   1:  PR[91,2] = PR[90,2] + -6.880;
   1:L PR[91] R[100]mm/sec CNT100;
   1:  PR[91,1] = PR[90,1] + -40.976;
   1:  PR[91,2] = PR[90,2] + -9.031;
   1:L PR[91] R[100]mm/sec CNT100;
   1:  PR[91,1] = PR[90,1] + -40.215;
   1:  PR[91,2] = PR[90,2] + -10.350;
   1:L PR[91] R[100]mm/sec CNT100;
   1:  PR[91,1] = PR[90,1] + -38.856;
   1:  PR[91,2] = PR[90,2] + -12.292;
   1:L PR[91] R[100]mm/sec CNT100;
   1:  PR[91,1] = PR[90,1] + -37.178;
   1:  PR[91,2] = PR[90,2] + -13.971;
   1:L PR[91] R[100]mm/sec CNT100;
   1:  PR[91,1] = PR[90,1] + -36.012;
   1:  PR[91,2] = PR[90,2] + -14.949;
   1:L PR[91] R[100]mm/sec CNT100;
   1:  PR[91,1] = PR[90,1] + -34.070;
   1:  PR[91,2] = PR[90,2] + -16.309;
   1:L PR[91] R[100]mm/sec CNT100;
   1:  PR[91,1] = PR[90,1] + -31.919;
   1:  PR[91,2] = PR[90,2] + -17.313;
   1:L PR[91] R[100]mm/sec CNT100;
   1:  PR[91,1] = PR[90,1] + -30.489;
   1:  PR[91,2] = PR[90,2] + -17.834;
   1:L PR[91] R[100]mm/sec CNT100;
   1:  PR[91,1] = PR[90,1] + -28.198;
   1:  PR[91,2] = PR[90,2] + -18.448;
   1:L PR[91] R[100]mm/sec CNT100;
   1:  PR[91,1] = PR[90,1] + -25.833;
   1:  PR[91,2] = PR[90,2] + -18.655;
   1:L PR[91] R[100]mm/sec CNT100;
   1:  PR[91,1] = PR[90,1] + -24.309;
   1:L PR[91] R[100]mm/sec CNT100;
   1:  PR[91,1] = PR[90,1] + -22.033;
   1:  PR[91,2] = PR[90,2] + -18.456;
   1:L PR[91] R[100]mm/sec CNT100;
   1:  PR[91,1] = PR[90,1] + -20.603;
   1:  PR[91,2] = PR[90,2] + -17.935;
   1:L PR[91] R[100]mm/sec CNT100;
   1:  PR[91,1] = PR[90,1] + -18.143;
   1:  PR[91,2] = PR[90,2] + -17.276;
   1:L PR[91] R[100]mm/sec CNT100;
   1:  PR[91,1] = PR[90,1] + -16.152;
   1:  PR[91,2] = PR[90,2] + -16.347;
   1:L PR[91] R[100]mm/sec CNT100;
   1:  PR[91,1] = PR[90,1] + -14.987;
   1:  PR[91,2] = PR[90,2] + -15.369;
   1:L PR[91] R[100]mm/sec CNT100;
   1:  PR[91,1] = PR[90,1] + -12.902;
   1:  PR[91,2] = PR[90,2] + -13.909;
   1:L PR[91] R[100]mm/sec CNT100;
   1:  PR[91,1] = PR[90,1] + -11.349;
   1:  PR[91,2] = PR[90,2] + -12.355;
   1:L PR[91] R[100]mm/sec CNT100;
   1:  PR[91,1] = PR[90,1] + -10.588;
   1:  PR[91,2] = PR[90,2] + -11.038;
   1:L PR[91] R[100]mm/sec CNT100;
   1:  PR[91,1] = PR[90,1] + -9.128;
   1:  PR[91,2] = PR[90,2] + -8.953;
   1:L PR[91] R[100]mm/sec CNT100;
   1:  PR[91,1] = PR[90,1] + -8.200;
   1:  PR[91,2] = PR[90,2] + -6.961;
   1:L PR[91] R[100]mm/sec CNT100;
   1:  PR[91,1] = PR[90,1] + -7.935;
   1:  PR[91,2] = PR[90,2] + -5.462;
   1:L PR[91] R[100]mm/sec CNT100;
   1:  PR[91,1] = PR[90,1] + -7.277;
   1:  PR[91,2] = PR[90,2] + -3.003;
   1:L PR[91] R[100]mm/sec CNT100;
   1:  PR[91,1] = PR[90,1] + -7.086;
   1:  PR[91,2] = PR[90,2] + -0.818;
   1:L PR[91] R[100]mm/sec CNT100;
   1:  PR[91,1] = PR[90,1] + -7.350;
   1:  PR[91,2] = PR[90,2] + 0.681;
   1:L PR[91] R[100]mm/sec CNT100;
   1:  PR[91,1] = PR[90,1] + -7.572;
   1:  PR[91,2] = PR[90,2] + 3.215;
   1:L PR[91] R[100]mm/sec CNT100;
   1:  PR[91,1] = PR[90,1] + -8.162;
   1:  PR[91,2] = PR[90,2] + 5.422;
   1:L PR[91] R[100]mm/sec CNT100;
   1:  PR[91,1] = PR[90,1] + -9.165;
   1:  PR[91,2] = PR[90,2] + 7.572;
   1:L PR[91] R[100]mm/sec CNT100;
   1:  PR[91,1] = PR[90,1] + -9.926;
   1:  PR[91,2] = PR[90,2] + 8.891;
   1:L PR[91] R[100]mm/sec CNT100;
   1:  PR[91,1] = PR[90,1] + -11.286;
   1:  PR[91,2] = PR[90,2] + 10.833;
   1:L PR[91] R[100]mm/sec CNT100;
   1:  PR[91,1] = PR[90,1] + -12.964;
   1:  PR[91,2] = PR[90,2] + 12.512;
   1:L PR[91] R[100]mm/sec CNT100;
   1:  PR[91,1] = PR[90,1] + -14.129;
   1:  PR[91,2] = PR[90,2] + 13.490;
   1:L PR[91] R[100]mm/sec CNT100;
   1:  PR[91,1] = PR[90,1] + -16.071;
   1:  PR[91,2] = PR[90,2] + 14.850;
   1:L PR[91] R[100]mm/sec CNT100;
   1:  PR[91,1] = PR[90,1] + -18.222;
   1:  PR[91,2] = PR[90,2] + 15.854;
   1:L PR[91] R[100]mm/sec CNT100;
   1:  PR[91,1] = PR[90,1] + -19.653;
   1:  PR[91,2] = PR[90,2] + 16.375;
   1:L PR[91] R[100]mm/sec CNT100;
   1:  PR[91,1] = PR[90,1] + -21.944;
   1:  PR[91,2] = PR[90,2] + 16.989;
   1:L PR[91] R[100]mm/sec CNT100;
   1:  PR[91,1] = PR[90,1] + -24.308;
   1:  PR[91,2] = PR[90,2] + 17.196;
   1:L PR[91] R[100]mm/sec CNT100;
   1:  PR[91,1] = PR[90,1] + -25.832;
   1:L PR[91] R[100]mm/sec CNT100;
   1:  PR[91,1] = PR[90,1] + -28.109;
   1:  PR[91,2] = PR[90,2] + 16.997;
   1:L PR[91] R[100]mm/sec CNT100;
   1:  PR[91,1] = PR[90,1] + -29.538;
   1:  PR[91,2] = PR[90,2] + 16.476;
   1:L PR[91] R[100]mm/sec CNT100;
   1:  PR[91,1] = PR[90,1] + -31.998;
   1:  PR[91,2] = PR[90,2] + 15.817;
   1:L PR[91] R[100]mm/sec CNT100;
   1:  PR[91,1] = PR[90,1] + -33.989;
   1:  PR[91,2] = PR[90,2] + 14.888;
   1:L PR[91] R[100]mm/sec CNT100;
   1:  PR[91,1] = PR[90,1] + -35.154;
   1:  PR[91,2] = PR[90,2] + 13.911;
   1:L PR[91] R[100]mm/sec CNT100;
   1:  PR[91,1] = PR[90,1] + -37.239;
   1:  PR[91,2] = PR[90,2] + 12.451;
   1:L PR[91] R[100]mm/sec CNT100;
   1:  PR[91,1] = PR[90,1] + -38.793;
   1:  PR[91,2] = PR[90,2] + 10.896;
   1:L PR[91] R[100]mm/sec CNT100;
   1:  PR[91,1] = PR[90,1] + -39.553;
   1:  PR[91,2] = PR[90,2] + 9.579;
   1:L PR[91] R[100]mm/sec CNT100;
   1:  PR[91,1] = PR[90,1] + -41.013;
   1:  PR[91,2] = PR[90,2] + 7.494;
   1:L PR[91] R[100]mm/sec CNT100;
   1:  PR[91,1] = PR[90,1] + -41.941;
   1:  PR[91,2] = PR[90,2] + 5.502;
   1:L PR[91] R[100]mm/sec CNT100;
   1:  PR[91,1] = PR[90,1] + -42.206;
   1:  PR[91,2] = PR[90,2] + 4.003;
   1:L PR[91] R[100]mm/sec CNT100;
   1:  PR[91,1] = PR[90,1] + -42.864;
   1:  PR[91,2] = PR[90,2] + 1.544;
   1:L PR[91] R[100]mm/sec CNT100;
   1:  PR[91,1] = PR[90,1] + -43.055;
   1:  PR[91,2] = PR[90,2] + -0.641;
   1:L PR[91] R[100]mm/sec CNT100;
   1:  PR[91,1] = PR[90,1] + -42.791;
   1:  PR[91,2] = PR[90,2] + -2.140;
   1:L PR[91] R[100]mm/sec CNT100TB   .50sec,CALL END_PUD;
   1:  PR[92] = PR[91];
   1:  PR[92,3] = PR[92,3] + 20;
   1:J PR[92] 10% FINE;
   1:  PR[91,1] = PR[90,1] + 29.399;
   1:  PR[91,2] = PR[90,2] + -17.935;
   1:  PR[92] = PR[91];
   1:  PR[92,3] = PR[92,3] + 20;
   1:J PR[92] 10% FINE;
   1:L PR[91] R[100]mm/sec CNT100;
   1:  CALL LASER_DRAHT_START;
   1:  PR[91,1] = PR[90,1] + 31.859;
   1:  PR[91,2] = PR[90,2] + -17.275;
   1:L PR[91] R[100]mm/sec CNT100;
   1:  PR[91,1] = PR[90,1] + 33.925;
   1:  PR[91,2] = PR[90,2] + -16.311;
   1:L PR[91] R[100]mm/sec CNT100;
   1:  PR[91,1] = PR[90,1] + 35.871;
   1:  PR[91,2] = PR[90,2] + -14.949;
   1:L PR[91] R[100]mm/sec CNT100;
   1:  PR[91,1] = PR[90,1] + 37.037;
   1:  PR[91,2] = PR[90,2] + -13.970;
   1:L PR[91] R[100]mm/sec CNT100;
   1:  PR[91,1] = PR[90,1] + 38.711;
   1:  PR[91,2] = PR[90,2] + -12.296;
   1:L PR[91] R[100]mm/sec CNT100;
   1:  PR[91,1] = PR[90,1] + 40.074;
   1:  PR[91,2] = PR[90,2] + -10.349;
   1:L PR[91] R[100]mm/sec CNT100;
   1:  PR[91,1] = PR[90,1] + 40.835;
   1:  PR[91,2] = PR[90,2] + -9.031;
   1:L PR[91] R[100]mm/sec CNT100;
   1:  PR[91,1] = PR[90,1] + 41.799;
   1:  PR[91,2] = PR[90,2] + -6.963;
   1:L PR[91] R[100]mm/sec CNT100;
   1:  PR[91,1] = PR[90,1] + 42.064;
   1:  PR[91,2] = PR[90,2] + -5.465;
   1:L PR[91] R[100]mm/sec CNT100;
   1:  PR[91,1] = PR[90,1] + 42.723;
   1:  PR[91,2] = PR[90,2] + -3.002;
   1:L PR[91] R[100]mm/sec CNT100;
   1:  PR[91,1] = PR[90,1] + 42.914;
   1:  PR[91,2] = PR[90,2] + -0.818;
   1:L PR[91] R[100]mm/sec CNT100;
   1:  PR[91,1] = PR[90,1] + 42.650;
   1:  PR[91,2] = PR[90,2] + 0.681;
   1:L PR[91] R[100]mm/sec CNT100;
   1:  PR[91,1] = PR[90,1] + 42.428;
   1:  PR[91,2] = PR[90,2] + 3.215;
   1:L PR[91] R[100]mm/sec CNT100;
   1:  PR[91,1] = PR[90,1] + 41.859;
   1:  PR[91,2] = PR[90,2] + 5.341;
   1:L PR[91] R[100]mm/sec CNT100;
   1:  PR[91,1] = PR[90,1] + 41.098;
   1:  PR[91,2] = PR[90,2] + 6.658;
   1:L PR[91] R[100]mm/sec CNT100;
   1:  PR[91,1] = PR[90,1] + 40.022;
   1:  PR[91,2] = PR[90,2] + 8.965;
   1:L PR[91] R[100]mm/sec CNT100;
   1:  PR[91,1] = PR[90,1] + 38.759;
   1:  PR[91,2] = PR[90,2] + 10.768;
   1:L PR[91] R[100]mm/sec CNT100;
   1:  PR[91,1] = PR[90,1] + 37.594;
   1:  PR[91,2] = PR[90,2] + 11.746;
   1:L PR[91] R[100]mm/sec CNT100;
   1:  PR[91,1] = PR[90,1] + 35.795;
   1:  PR[91,2] = PR[90,2] + 13.543;
   1:L PR[91] R[100]mm/sec CNT100;
   1:  PR[91,1] = PR[90,1] + 33.992;
   1:  PR[91,2] = PR[90,2] + 14.805;
   1:L PR[91] R[100]mm/sec CNT100;
   1:  PR[91,1] = PR[90,1] + 32.563;
   1:  PR[91,2] = PR[90,2] + 15.325;
   1:L PR[91] R[100]mm/sec CNT100;
   1:  PR[91,1] = PR[90,1] + 30.258;
   1:  PR[91,2] = PR[90,2] + 16.399;
   1:L PR[91] R[100]mm/sec CNT100;
   1:  PR[91,1] = PR[90,1] + 28.134;
   1:  PR[91,2] = PR[90,2] + 16.968;
   1:L PR[91] R[100]mm/sec CNT100;
   1:  PR[91,1] = PR[90,1] + 26.611;
   1:L PR[91] R[100]mm/sec CNT100;
   1:  PR[91,1] = PR[90,1] + 24.075;
   1:  PR[91,2] = PR[90,2] + 17.189;
   1:L PR[91] R[100]mm/sec CNT100;
   1:  PR[91,1] = PR[90,1] + 21.889;
   1:  PR[91,2] = PR[90,2] + 16.997;
   1:L PR[91] R[100]mm/sec CNT100;
   1:  PR[91,1] = PR[90,1] + 20.460;
   1:  PR[91,2] = PR[90,2] + 16.476;
   1:L PR[91] R[100]mm/sec CNT100;
   1:  PR[91,1] = PR[90,1] + 17.999;
   1:  PR[91,2] = PR[90,2] + 15.816;
   1:L PR[91] R[100]mm/sec CNT100;
   1:  PR[91,1] = PR[90,1] + 15.933;
   1:  PR[91,2] = PR[90,2] + 14.852;
   1:L PR[91] R[100]mm/sec CNT100;
   1:  PR[91,1] = PR[90,1] + 13.988;
   1:  PR[91,2] = PR[90,2] + 13.490;
   1:L PR[91] R[100]mm/sec CNT100;
   1:  PR[91,1] = PR[90,1] + 12.822;
   1:  PR[91,2] = PR[90,2] + 12.512;
   1:L PR[91] R[100]mm/sec CNT100;
   1:  PR[91,1] = PR[90,1] + 11.148;
   1:  PR[91,2] = PR[90,2] + 10.838;
   1:L PR[91] R[100]mm/sec CNT100;
   1:  PR[91,1] = PR[90,1] + 9.785;
   1:  PR[91,2] = PR[90,2] + 8.891;
   1:L PR[91] R[100]mm/sec CNT100;
   1:  PR[91,1] = PR[90,1] + 9.024;
   1:  PR[91,2] = PR[90,2] + 7.572;
   1:L PR[91] R[100]mm/sec CNT100;
   1:  PR[91,1] = PR[90,1] + 8.060;
   1:  PR[91,2] = PR[90,2] + 5.505;
   1:L PR[91] R[100]mm/sec CNT100;
   1:  PR[91,1] = PR[90,1] + 7.795;
   1:  PR[91,2] = PR[90,2] + 4.006;
   1:L PR[91] R[100]mm/sec CNT100;
   1:  PR[91,1] = PR[90,1] + 7.136;
   1:  PR[91,2] = PR[90,2] + 1.543;
   1:L PR[91] R[100]mm/sec CNT100;
   1:  PR[91,1] = PR[90,1] + 6.945;
   1:  PR[91,2] = PR[90,2] + -0.641;
   1:L PR[91] R[100]mm/sec CNT100;
   1:  PR[91,1] = PR[90,1] + 7.209;
   1:  PR[91,2] = PR[90,2] + -2.140;
   1:L PR[91] R[100]mm/sec CNT100;
   1:  PR[91,1] = PR[90,1] + 7.431;
   1:  PR[91,2] = PR[90,2] + -4.674;
   1:L PR[91] R[100]mm/sec CNT100;
   1:  PR[91,1] = PR[90,1] + 8.000;
   1:  PR[91,2] = PR[90,2] + -6.799;
   1:L PR[91] R[100]mm/sec CNT100;
   1:  PR[91,1] = PR[90,1] + 8.761;
   1:  PR[91,2] = PR[90,2] + -8.116;
   1:L PR[91] R[100]mm/sec CNT100;
   1:  PR[91,1] = PR[90,1] + 9.837;
   1:  PR[91,2] = PR[90,2] + -10.424;
   1:L PR[91] R[100]mm/sec CNT100;
   1:  PR[91,1] = PR[90,1] + 11.100;
   1:  PR[91,2] = PR[90,2] + -12.227;
   1:L PR[91] R[100]mm/sec CNT100;
   1:  PR[91,1] = PR[90,1] + 12.265;
   1:  PR[91,2] = PR[90,2] + -13.205;
   1:L PR[91] R[100]mm/sec CNT100;
   1:  PR[91,1] = PR[90,1] + 14.064;
   1:  PR[91,2] = PR[90,2] + -15.002;
   1:L PR[91] R[100]mm/sec CNT100;
   1:  PR[91,1] = PR[90,1] + 15.866;
   1:  PR[91,2] = PR[90,2] + -16.264;
   1:L PR[91] R[100]mm/sec CNT100;
   1:  PR[91,1] = PR[90,1] + 17.296;
   1:  PR[91,2] = PR[90,2] + -16.784;
   1:L PR[91] R[100]mm/sec CNT100;
   1:  PR[91,1] = PR[90,1] + 19.601;
   1:  PR[91,2] = PR[90,2] + -17.858;
   1:L PR[91] R[100]mm/sec CNT100;
   1:  PR[91,1] = PR[90,1] + 21.725;
   1:  PR[91,2] = PR[90,2] + -18.427;
   1:L PR[91] R[100]mm/sec CNT100;
   1:  PR[91,1] = PR[90,1] + 23.247;
   1:L PR[91] R[100]mm/sec CNT100;
   1:  PR[91,1] = PR[90,1] + 25.783;
   1:  PR[91,2] = PR[90,2] + -18.647;
   1:L PR[91] R[100]mm/sec CNT100;
   1:  PR[91,1] = PR[90,1] + 27.970;
   1:  PR[91,2] = PR[90,2] + -18.455;
   1:L PR[91] R[100]mm/sec CNT100;
   1:  PR[91,1] = PR[90,1] + 29.399;
   1:  PR[91,2] = PR[90,2] + -17.935;
   1:L PR[91] R[100]mm/sec CNT100TB   .50sec,CALL END_PUD;
   1:  PR[92] = PR[91];
   1:  PR[92,3] = PR[92,3] + 20;
   1:J PR[92] 10% FINE;
   1:  PR[91,1] = PR[90,1] + 92.914;
   1:  PR[91,2] = PR[90,2] + -0.818;
   1:  PR[92] = PR[91];
   1:  PR[92,3] = PR[92,3] + 20;
   1:J PR[92] 10% FINE;
   1:L PR[91] R[100]mm/sec CNT100;
   1:  CALL LASER_DRAHT_START;
   1:  PR[91,1] = PR[90,1] + 92.650;
   1:  PR[91,2] = PR[90,2] + 0.681;
   1:L PR[91] R[100]mm/sec CNT100;
   1:  PR[91,1] = PR[90,1] + 92.428;
   1:  PR[91,2] = PR[90,2] + 3.215;
   1:L PR[91] R[100]mm/sec CNT100;
   1:  PR[91,1] = PR[90,1] + 91.836;
   1:  PR[91,2] = PR[90,2] + 5.425;
   1:L PR[91] R[100]mm/sec CNT100;
   1:  PR[91,1] = PR[90,1] + 90.835;
   1:  PR[91,2] = PR[90,2] + 7.572;
   1:L PR[91] R[100]mm/sec CNT100;
   1:  PR[91,1] = PR[90,1] + 90.074;
   1:  PR[91,2] = PR[90,2] + 8.891;
   1:L PR[91] R[100]mm/sec CNT100;
   1:  PR[91,1] = PR[90,1] + 88.761;
   1:  PR[91,2] = PR[90,2] + 10.765;
   1:L PR[91] R[100]mm/sec CNT100;
   1:  PR[91,1] = PR[90,1] + 87.596;
   1:  PR[91,2] = PR[90,2] + 11.743;
   1:L PR[91] R[100]mm/sec CNT100;
   1:  PR[91,1] = PR[90,1] + 85.799;
   1:  PR[91,2] = PR[90,2] + 13.540;
   1:L PR[91] R[100]mm/sec CNT100;
   1:  PR[91,1] = PR[90,1] + 83.998;
   1:  PR[91,2] = PR[90,2] + 14.802;
   1:L PR[91] R[100]mm/sec CNT100;
   1:  PR[91,1] = PR[90,1] + 82.568;
   1:  PR[91,2] = PR[90,2] + 15.322;
   1:L PR[91] R[100]mm/sec CNT100;
   1:  PR[91,1] = PR[90,1] + 80.265;
   1:  PR[91,2] = PR[90,2] + 16.397;
   1:L PR[91] R[100]mm/sec CNT100;
   1:  PR[91,1] = PR[90,1] + 78.058;
   1:  PR[91,2] = PR[90,2] + 16.989;
   1:L PR[91] R[100]mm/sec CNT100;
   1:  PR[91,1] = PR[90,1] + 75.697;
   1:  PR[91,2] = PR[90,2] + 17.196;
   1:L PR[91] R[100]mm/sec CNT100;
   1:  PR[91,1] = PR[90,1] + 74.173;
   1:L PR[91] R[100]mm/sec CNT100;
   1:  PR[91,1] = PR[90,1] + 71.810;
   1:  PR[91,2] = PR[90,2] + 16.990;
   1:L PR[91] R[100]mm/sec CNT100;
   1:  PR[91,1] = PR[90,1] + 69.517;
   1:  PR[91,2] = PR[90,2] + 16.377;
   1:L PR[91] R[100]mm/sec CNT100;
   1:  PR[91,1] = PR[90,1] + 68.086;
   1:  PR[91,2] = PR[90,2] + 15.856;
   1:L PR[91] R[100]mm/sec CNT100;
   1:  PR[91,1] = PR[90,1] + 65.938;
   1:  PR[91,2] = PR[90,2] + 14.855;
   1:L PR[91] R[100]mm/sec CNT100;
   1:  PR[91,1] = PR[90,1] + 63.992;
   1:  PR[91,2] = PR[90,2] + 13.493;
   1:L PR[91] R[100]mm/sec CNT100;
   1:  PR[91,1] = PR[90,1] + 62.826;
   1:  PR[91,2] = PR[90,2] + 12.515;
   1:L PR[91] R[100]mm/sec CNT100;
   1:  PR[91,1] = PR[90,1] + 61.151;
   1:  PR[91,2] = PR[90,2] + 10.840;
   1:L PR[91] R[100]mm/sec CNT100;
   1:  PR[91,1] = PR[90,1] + 59.786;
   1:  PR[91,2] = PR[90,2] + 8.893;
   1:L PR[91] R[100]mm/sec CNT100;
   1:  PR[91,1] = PR[90,1] + 59.025;
   1:  PR[91,2] = PR[90,2] + 7.575;
   1:L PR[91] R[100]mm/sec CNT100;
   1:  PR[91,1] = PR[90,1] + 58.023;
   1:  PR[91,2] = PR[90,2] + 5.426;
   1:L PR[91] R[100]mm/sec CNT100;
   1:  PR[91,1] = PR[90,1] + 57.408;
   1:  PR[91,2] = PR[90,2] + 3.130;
   1:L PR[91] R[100]mm/sec CNT100;
   1:  PR[91,1] = PR[90,1] + 57.143;
   1:  PR[91,2] = PR[90,2] + 1.630;
   1:L PR[91] R[100]mm/sec CNT100;
   1:  PR[91,1] = PR[90,1] + 56.945;
   1:  PR[91,2] = PR[90,2] + -0.641;
   1:L PR[91] R[100]mm/sec CNT100;
   1:  PR[91,1] = PR[90,1] + 57.209;
   1:  PR[91,2] = PR[90,2] + -2.140;
   1:L PR[91] R[100]mm/sec CNT100;
   1:  PR[91,1] = PR[90,1] + 57.431;
   1:  PR[91,2] = PR[90,2] + -4.674;
   1:L PR[91] R[100]mm/sec CNT100;
   1:  PR[91,1] = PR[90,1] + 58.022;
   1:  PR[91,2] = PR[90,2] + -6.884;
   1:L PR[91] R[100]mm/sec CNT100;
   1:  PR[91,1] = PR[90,1] + 59.024;
   1:  PR[91,2] = PR[90,2] + -9.031;
   1:L PR[91] R[100]mm/sec CNT100;
   1:  PR[91,1] = PR[90,1] + 59.785;
   1:  PR[91,2] = PR[90,2] + -10.349;
   1:L PR[91] R[100]mm/sec CNT100;
   1:  PR[91,1] = PR[90,1] + 61.098;
   1:  PR[91,2] = PR[90,2] + -12.224;
   1:L PR[91] R[100]mm/sec CNT100;
   1:  PR[91,1] = PR[90,1] + 62.262;
   1:  PR[91,2] = PR[90,2] + -13.202;
   1:L PR[91] R[100]mm/sec CNT100;
   1:  PR[91,1] = PR[90,1] + 64.060;
   1:  PR[91,2] = PR[90,2] + -14.999;
   1:L PR[91] R[100]mm/sec CNT100;
   1:  PR[91,1] = PR[90,1] + 65.861;
   1:  PR[91,2] = PR[90,2] + -16.261;
   1:L PR[91] R[100]mm/sec CNT100;
   1:  PR[91,1] = PR[90,1] + 67.291;
   1:  PR[91,2] = PR[90,2] + -16.781;
   1:L PR[91] R[100]mm/sec CNT100;
   1:  PR[91,1] = PR[90,1] + 69.594;
   1:  PR[91,2] = PR[90,2] + -17.856;
   1:L PR[91] R[100]mm/sec CNT100;
   1:  PR[91,1] = PR[90,1] + 71.801;
   1:  PR[91,2] = PR[90,2] + -18.448;
   1:L PR[91] R[100]mm/sec CNT100;
   1:  PR[91,1] = PR[90,1] + 74.162;
   1:  PR[91,2] = PR[90,2] + -18.655;
   1:L PR[91] R[100]mm/sec CNT100;
   1:  PR[91,1] = PR[90,1] + 75.686;
   1:L PR[91] R[100]mm/sec CNT100;
   1:  PR[91,1] = PR[90,1] + 78.049;
   1:  PR[91,2] = PR[90,2] + -18.449;
   1:L PR[91] R[100]mm/sec CNT100;
   1:  PR[91,1] = PR[90,1] + 80.342;
   1:  PR[91,2] = PR[90,2] + -17.836;
   1:L PR[91] R[100]mm/sec CNT100;
   1:  PR[91,1] = PR[90,1] + 81.773;
   1:  PR[91,2] = PR[90,2] + -17.315;
   1:L PR[91] R[100]mm/sec CNT100;
   1:  PR[91,1] = PR[90,1] + 83.920;
   1:  PR[91,2] = PR[90,2] + -16.314;
   1:L PR[91] R[100]mm/sec CNT100;
   1:  PR[91,1] = PR[90,1] + 85.867;
   1:  PR[91,2] = PR[90,2] + -14.952;
   1:L PR[91] R[100]mm/sec CNT100;
   1:  PR[91,1] = PR[90,1] + 87.033;
   1:  PR[91,2] = PR[90,2] + -13.974;
   1:L PR[91] R[100]mm/sec CNT100;
   1:  PR[91,1] = PR[90,1] + 88.708;
   1:  PR[91,2] = PR[90,2] + -12.299;
   1:L PR[91] R[100]mm/sec CNT100;
   1:  PR[91,1] = PR[90,1] + 90.073;
   1:  PR[91,2] = PR[90,2] + -10.352;
   1:L PR[91] R[100]mm/sec CNT100;
   1:  PR[91,1] = PR[90,1] + 90.834;
   1:  PR[91,2] = PR[90,2] + -9.034;
   1:L PR[91] R[100]mm/sec CNT100;
   1:  PR[91,1] = PR[90,1] + 91.836;
   1:  PR[91,2] = PR[90,2] + -6.885;
   1:L PR[91] R[100]mm/sec CNT100;
   1:  PR[91,1] = PR[90,1] + 92.451;
   1:  PR[91,2] = PR[90,2] + -4.589;
   1:L PR[91] R[100]mm/sec CNT100;
   1:  PR[91,1] = PR[90,1] + 92.716;
   1:  PR[91,2] = PR[90,2] + -3.089;
   1:L PR[91] R[100]mm/sec CNT100;
   1:  PR[91,1] = PR[90,1] + 92.914;
   1:  PR[91,2] = PR[90,2] + -0.818;
   1:L PR[91] R[100]mm/sec CNT100TB   .50sec,CALL END_PUD;
   1:  PR[92] = PR[91];
   1:  PR[92,3] = PR[92,3] + 20;
   1:J PR[92] 10% FINE;
   1:  PR[91] = PR[90];
   1:  PR[91,1] = PR[90,1] + -78.273;
   1:  PR[91,2] = PR[90,2] + -18.427;
   1:  PR[91,3] = PR[90,3] + 7.995;
   1:  PR[92] = PR[91];
   1:  PR[92,3] = PR[92,3] + 20;
   1:J PR[92] 10% FINE;
   1:L PR[91] R[100]mm/sec CNT100;
   1:  CALL LASER_DRAHT_START;
   1:  PR[91,1] = PR[90,1] + -77.880;
   1:L PR[91] R[100]mm/sec CNT100;
   1:  PR[91,1] = PR[90,1] + -74.780;
   1:  PR[91,2] = PR[90,2] + -18.697;
   1:L PR[91] R[100]mm/sec CNT100;
   1:  PR[91,1] = PR[90,1] + -72.030;
   1:  PR[91,2] = PR[90,2] + -18.455;
   1:L PR[91] R[100]mm/sec CNT100;
   1:  PR[91,1] = PR[90,1] + -71.661;
   1:  PR[91,2] = PR[90,2] + -18.321;
   1:L PR[91] R[100]mm/sec CNT100;
   1:  PR[91,1] = PR[90,1] + -68.653;
   1:  PR[91,2] = PR[90,2] + -17.514;
   1:L PR[91] R[100]mm/sec CNT100;
   1:  PR[91,1] = PR[90,1] + -66.075;
   1:  PR[91,2] = PR[90,2] + -16.311;
   1:L PR[91] R[100]mm/sec CNT100;
   1:  PR[91,1] = PR[90,1] + -63.665;
   1:  PR[91,2] = PR[90,2] + -14.624;
   1:L PR[91] R[100]mm/sec CNT100;
   1:  PR[91,1] = PR[90,1] + -63.363;
   1:  PR[91,2] = PR[90,2] + -14.371;
   1:L PR[91] R[100]mm/sec CNT100;
   1:  PR[91,1] = PR[90,1] + -61.289;
   1:  PR[91,2] = PR[90,2] + -12.297;
   1:L PR[91] R[100]mm/sec CNT100;
   1:  PR[91,1] = PR[90,1] + -59.601;
   1:  PR[91,2] = PR[90,2] + -9.885;
   1:L PR[91] R[100]mm/sec CNT100;
   1:  PR[91,1] = PR[90,1] + -59.404;
   1:  PR[91,2] = PR[90,2] + -9.544;
   1:L PR[91] R[100]mm/sec CNT100;
   1:  PR[91,1] = PR[90,1] + -58.201;
   1:  PR[91,2] = PR[90,2] + -6.963;
   1:L PR[91] R[100]mm/sec CNT100;
   1:  PR[91,1] = PR[90,1] + -58.132;
   1:  PR[91,2] = PR[90,2] + -6.576;
   1:L PR[91] R[100]mm/sec CNT100;
   1:  PR[91,1] = PR[90,1] + -57.326;
   1:  PR[91,2] = PR[90,2] + -3.565;
   1:L PR[91] R[100]mm/sec CNT100;
   1:  PR[91,1] = PR[90,1] + -57.086;
   1:  PR[91,2] = PR[90,2] + -0.818;
   1:L PR[91] R[100]mm/sec CNT100;
   1:  PR[91,1] = PR[90,1] + -57.154;
   1:  PR[91,2] = PR[90,2] + -0.430;
   1:L PR[91] R[100]mm/sec CNT100;
   1:  PR[91,1] = PR[90,1] + -57.425;
   1:  PR[91,2] = PR[90,2] + 2.667;
   1:L PR[91] R[100]mm/sec CNT100;
   1:  PR[91,1] = PR[90,1] + -58.141;
   1:  PR[91,2] = PR[90,2] + 5.341;
   1:L PR[91] R[100]mm/sec CNT100;
   1:  PR[91,1] = PR[90,1] + -58.337;
   1:  PR[91,2] = PR[90,2] + 5.680;
   1:L PR[91] R[100]mm/sec CNT100;
   1:  PR[91,1] = PR[90,1] + -59.653;
   1:  PR[91,2] = PR[90,2] + 8.501;
   1:L PR[91] R[100]mm/sec CNT100;
   1:  PR[91,1] = PR[90,1] + -61.242;
   1:  PR[91,2] = PR[90,2] + 10.769;
   1:L PR[91] R[100]mm/sec CNT100;
   1:  PR[91,1] = PR[90,1] + -61.543;
   1:  PR[91,2] = PR[90,2] + 11.022;
   1:L PR[91] R[100]mm/sec CNT100;
   1:  PR[91,1] = PR[90,1] + -63.742;
   1:  PR[91,2] = PR[90,2] + 13.219;
   1:L PR[91] R[100]mm/sec CNT100;
   1:  PR[91,1] = PR[90,1] + -66.009;
   1:  PR[91,2] = PR[90,2] + 14.806;
   1:L PR[91] R[100]mm/sec CNT100;
   1:  PR[91,1] = PR[90,1] + -66.378;
   1:  PR[91,2] = PR[90,2] + 14.940;
   1:L PR[91] R[100]mm/sec CNT100;
   1:  PR[91,1] = PR[90,1] + -69.196;
   1:  PR[91,2] = PR[90,2] + 16.253;
   1:L PR[91] R[100]mm/sec CNT100;
   1:  PR[91,1] = PR[90,1] + -71.868;
   1:  PR[91,2] = PR[90,2] + 16.968;
   1:L PR[91] R[100]mm/sec CNT100;
   1:  PR[91,1] = PR[90,1] + -72.261;
   1:L PR[91] R[100]mm/sec CNT100;
   1:  PR[91,1] = PR[90,1] + -75.361;
   1:  PR[91,2] = PR[90,2] + 17.238;
   1:L PR[91] R[100]mm/sec CNT100;
   1:  PR[91,1] = PR[90,1] + -78.111;
   1:  PR[91,2] = PR[90,2] + 16.997;
   1:L PR[91] R[100]mm/sec CNT100;
   1:  PR[91,1] = PR[90,1] + -78.480;
   1:  PR[91,2] = PR[90,2] + 16.862;
   1:L PR[91] R[100]mm/sec CNT100;
   1:  PR[91,1] = PR[90,1] + -81.488;
   1:  PR[91,2] = PR[90,2] + 16.055;
   1:L PR[91] R[100]mm/sec CNT100;
   1:  PR[91,1] = PR[90,1] + -84.066;
   1:  PR[91,2] = PR[90,2] + 14.853;
   1:L PR[91] R[100]mm/sec CNT100;
   1:  PR[91,1] = PR[90,1] + -86.476;
   1:  PR[91,2] = PR[90,2] + 13.165;
   1:L PR[91] R[100]mm/sec CNT100;
   1:  PR[91,1] = PR[90,1] + -86.778;
   1:  PR[91,2] = PR[90,2] + 12.912;
   1:L PR[91] R[100]mm/sec CNT100;
   1:  PR[91,1] = PR[90,1] + -88.852;
   1:  PR[91,2] = PR[90,2] + 10.838;
   1:L PR[91] R[100]mm/sec CNT100;
   1:  PR[91,1] = PR[90,1] + -90.540;
   1:  PR[91,2] = PR[90,2] + 8.426;
   1:L PR[91] R[100]mm/sec CNT100;
   1:  PR[91,1] = PR[90,1] + -90.737;
   1:  PR[91,2] = PR[90,2] + 8.085;
   1:L PR[91] R[100]mm/sec CNT100;
   1:  PR[91,1] = PR[90,1] + -91.941;
   1:  PR[91,2] = PR[90,2] + 5.504;
   1:L PR[91] R[100]mm/sec CNT100;
   1:  PR[91,1] = PR[90,1] + -92.009;
   1:  PR[91,2] = PR[90,2] + 5.117;
   1:L PR[91] R[100]mm/sec CNT100;
   1:  PR[91,1] = PR[90,1] + -92.815;
   1:  PR[91,2] = PR[90,2] + 2.107;
   1:L PR[91] R[100]mm/sec CNT100;
   1:  PR[91,1] = PR[90,1] + -93.055;
   1:  PR[91,2] = PR[90,2] + -0.641;
   1:L PR[91] R[100]mm/sec CNT100;
   1:  PR[91,1] = PR[90,1] + -92.987;
   1:  PR[91,2] = PR[90,2] + -1.028;
   1:L PR[91] R[100]mm/sec CNT100;
   1:  PR[91,1] = PR[90,1] + -92.716;
   1:  PR[91,2] = PR[90,2] + -4.126;
   1:L PR[91] R[100]mm/sec CNT100;
   1:  PR[91,1] = PR[90,1] + -92.000;
   1:  PR[91,2] = PR[90,2] + -6.799;
   1:L PR[91] R[100]mm/sec CNT100;
   1:  PR[91,1] = PR[90,1] + -91.804;
   1:  PR[91,2] = PR[90,2] + -7.139;
   1:L PR[91] R[100]mm/sec CNT100;
   1:  PR[91,1] = PR[90,1] + -90.488;
   1:  PR[91,2] = PR[90,2] + -9.960;
   1:L PR[91] R[100]mm/sec CNT100;
   1:  PR[91,1] = PR[90,1] + -88.899;
   1:  PR[91,2] = PR[90,2] + -12.228;
   1:L PR[91] R[100]mm/sec CNT100;
   1:  PR[91,1] = PR[90,1] + -88.599;
   1:  PR[91,2] = PR[90,2] + -12.480;
   1:L PR[91] R[100]mm/sec CNT100;
   1:  PR[91,1] = PR[90,1] + -86.400;
   1:  PR[91,2] = PR[90,2] + -14.678;
   1:L PR[91] R[100]mm/sec CNT100;
   1:  PR[91,1] = PR[90,1] + -84.132;
   1:  PR[91,2] = PR[90,2] + -16.265;
   1:L PR[91] R[100]mm/sec CNT100;
   1:  PR[91,1] = PR[90,1] + -83.763;
   1:  PR[91,2] = PR[90,2] + -16.399;
   1:L PR[91] R[100]mm/sec CNT100;
   1:  PR[91,1] = PR[90,1] + -80.945;
   1:  PR[91,2] = PR[90,2] + -17.712;
   1:L PR[91] R[100]mm/sec CNT100;
   1:  PR[91,1] = PR[90,1] + -78.273;
   1:  PR[91,2] = PR[90,2] + -18.427;
   1:L PR[91] R[100]mm/sec CNT100TB   .50sec,CALL END_PUD;
   1:  PR[92] = PR[91];
   1:  PR[92,3] = PR[92,3] + 20;
   1:J PR[92] 10% FINE;
   1:  PR[91,1] = PR[90,1] + -43.055;
   1:  PR[91,2] = PR[90,2] + -0.641;
   1:  PR[92] = PR[91];
   1:  PR[92,3] = PR[92,3] + 20;
   1:J PR[92] 10% FINE;
   1:L PR[91] R[100]mm/sec CNT100;
   1:  CALL LASER_DRAHT_START;
   1:  PR[91,1] = PR[90,1] + -42.987;
   1:  PR[91,2] = PR[90,2] + -1.028;
   1:L PR[91] R[100]mm/sec CNT100;
   1:  PR[91,1] = PR[90,1] + -42.716;
   1:  PR[91,2] = PR[90,2] + -4.126;
   1:L PR[91] R[100]mm/sec CNT100;
   1:  PR[91,1] = PR[90,1] + -41.979;
   1:  PR[91,2] = PR[90,2] + -6.879;
   1:L PR[91] R[100]mm/sec CNT100;
   1:  PR[91,1] = PR[90,1] + -40.737;
   1:  PR[91,2] = PR[90,2] + -9.544;
   1:L PR[91] R[100]mm/sec CNT100;
   1:  PR[91,1] = PR[90,1] + -40.540;
   1:  PR[91,2] = PR[90,2] + -9.885;
   1:L PR[91] R[100]mm/sec CNT100;
   1:  PR[91,1] = PR[90,1] + -38.856;
   1:  PR[91,2] = PR[90,2] + -12.291;
   1:L PR[91] R[100]mm/sec CNT100;
   1:  PR[91,1] = PR[90,1] + -36.778;
   1:  PR[91,2] = PR[90,2] + -14.371;
   1:L PR[91] R[100]mm/sec CNT100;
   1:  PR[91,1] = PR[90,1] + -36.476;
   1:  PR[91,2] = PR[90,2] + -14.624;
   1:L PR[91] R[100]mm/sec CNT100;
   1:  PR[91,1] = PR[90,1] + -34.071;
   1:  PR[91,2] = PR[90,2] + -16.309;
   1:L PR[91] R[100]mm/sec CNT100;
   1:  PR[91,1] = PR[90,1] + -31.406;
   1:  PR[91,2] = PR[90,2] + -17.552;
   1:L PR[91] R[100]mm/sec CNT100;
   1:  PR[91,1] = PR[90,1] + -31.036;
   1:  PR[91,2] = PR[90,2] + -17.687;
   1:L PR[91] R[100]mm/sec CNT100;
   1:  PR[91,1] = PR[90,1] + -28.198;
   1:  PR[91,2] = PR[90,2] + -18.448;
   1:L PR[91] R[100]mm/sec CNT100;
   1:  PR[91,1] = PR[90,1] + -25.268;
   1:  PR[91,2] = PR[90,2] + -18.704;
   1:L PR[91] R[100]mm/sec CNT100;
   1:  PR[91,1] = PR[90,1] + -24.874;
   1:L PR[91] R[100]mm/sec CNT100;
   1:  PR[91,1] = PR[90,1] + -22.033;
   1:  PR[91,2] = PR[90,2] + -18.456;
   1:L PR[91] R[100]mm/sec CNT100;
   1:  PR[91,1] = PR[90,1] + -21.664;
   1:  PR[91,2] = PR[90,2] + -18.321;
   1:L PR[91] R[100]mm/sec CNT100;
   1:  PR[91,1] = PR[90,1] + -18.657;
   1:  PR[91,2] = PR[90,2] + -17.515;
   1:L PR[91] R[100]mm/sec CNT100;
   1:  PR[91,1] = PR[90,1] + -16.152;
   1:  PR[91,2] = PR[90,2] + -16.347;
   1:L PR[91] R[100]mm/sec CNT100;
   1:  PR[91,1] = PR[90,1] + -15.851;
   1:  PR[91,2] = PR[90,2] + -16.095;
   1:L PR[91] R[100]mm/sec CNT100;
   1:  PR[91,1] = PR[90,1] + -13.303;
   1:  PR[91,2] = PR[90,2] + -14.310;
   1:L PR[91] R[100]mm/sec CNT100;
   1:  PR[91,1] = PR[90,1] + -11.348;
   1:  PR[91,2] = PR[90,2] + -12.355;
   1:L PR[91] R[100]mm/sec CNT100;
   1:  PR[91,1] = PR[90,1] + -11.152;
   1:  PR[91,2] = PR[90,2] + -12.015;
   1:L PR[91] R[100]mm/sec CNT100;
   1:  PR[91,1] = PR[90,1] + -9.367;
   1:  PR[91,2] = PR[90,2] + -9.466;
   1:L PR[91] R[100]mm/sec CNT100;
   1:  PR[91,1] = PR[90,1] + -8.199;
   1:  PR[91,2] = PR[90,2] + -6.960;
   1:L PR[91] R[100]mm/sec CNT100;
   1:  PR[91,1] = PR[90,1] + -8.131;
   1:  PR[91,2] = PR[90,2] + -6.573;
   1:L PR[91] R[100]mm/sec CNT100;
   1:  PR[91,1] = PR[90,1] + -7.326;
   1:  PR[91,2] = PR[90,2] + -3.567;
   1:L PR[91] R[100]mm/sec CNT100;
   1:  PR[91,1] = PR[90,1] + -7.086;
   1:  PR[91,2] = PR[90,2] + -0.818;
   1:L PR[91] R[100]mm/sec CNT100;
   1:  PR[91,1] = PR[90,1] + -7.154;
   1:  PR[91,2] = PR[90,2] + -0.430;
   1:L PR[91] R[100]mm/sec CNT100;
   1:  PR[91,1] = PR[90,1] + -7.425;
   1:  PR[91,2] = PR[90,2] + 2.667;
   1:L PR[91] R[100]mm/sec CNT100;
   1:  PR[91,1] = PR[90,1] + -8.162;
   1:  PR[91,2] = PR[90,2] + 5.420;
   1:L PR[91] R[100]mm/sec CNT100;
   1:  PR[91,1] = PR[90,1] + -9.404;
   1:  PR[91,2] = PR[90,2] + 8.085;
   1:L PR[91] R[100]mm/sec CNT100;
   1:  PR[91,1] = PR[90,1] + -9.601;
   1:  PR[91,2] = PR[90,2] + 8.426;
   1:L PR[91] R[100]mm/sec CNT100;
   1:  PR[91,1] = PR[90,1] + -11.285;
   1:  PR[91,2] = PR[90,2] + 10.833;
   1:L PR[91] R[100]mm/sec CNT100;
   1:  PR[91,1] = PR[90,1] + -13.364;
   1:  PR[91,2] = PR[90,2] + 12.912;
   1:L PR[91] R[100]mm/sec CNT100;
   1:  PR[91,1] = PR[90,1] + -13.665;
   1:  PR[91,2] = PR[90,2] + 13.165;
   1:L PR[91] R[100]mm/sec CNT100;
   1:  PR[91,1] = PR[90,1] + -16.070;
   1:  PR[91,2] = PR[90,2] + 14.850;
   1:L PR[91] R[100]mm/sec CNT100;
   1:  PR[91,1] = PR[90,1] + -18.735;
   1:  PR[91,2] = PR[90,2] + 16.093;
   1:L PR[91] R[100]mm/sec CNT100;
   1:  PR[91,1] = PR[90,1] + -19.105;
   1:  PR[91,2] = PR[90,2] + 16.228;
   1:L PR[91] R[100]mm/sec CNT100;
   1:  PR[91,1] = PR[90,1] + -21.943;
   1:  PR[91,2] = PR[90,2] + 16.989;
   1:L PR[91] R[100]mm/sec CNT100;
   1:  PR[91,1] = PR[90,1] + -24.873;
   1:  PR[91,2] = PR[90,2] + 17.246;
   1:L PR[91] R[100]mm/sec CNT100;
   1:  PR[91,1] = PR[90,1] + -25.267;
   1:L PR[91] R[100]mm/sec CNT100;
   1:  PR[91,1] = PR[90,1] + -28.109;
   1:  PR[91,2] = PR[90,2] + 16.997;
   1:L PR[91] R[100]mm/sec CNT100;
   1:  PR[91,1] = PR[90,1] + -28.477;
   1:  PR[91,2] = PR[90,2] + 16.863;
   1:L PR[91] R[100]mm/sec CNT100;
   1:  PR[91,1] = PR[90,1] + -31.485;
   1:  PR[91,2] = PR[90,2] + 16.057;
   1:L PR[91] R[100]mm/sec CNT100;
   1:  PR[91,1] = PR[90,1] + -33.990;
   1:  PR[91,2] = PR[90,2] + 14.888;
   1:L PR[91] R[100]mm/sec CNT100;
   1:  PR[91,1] = PR[90,1] + -34.290;
   1:  PR[91,2] = PR[90,2] + 14.636;
   1:L PR[91] R[100]mm/sec CNT100;
   1:  PR[91,1] = PR[90,1] + -36.838;
   1:  PR[91,2] = PR[90,2] + 12.851;
   1:L PR[91] R[100]mm/sec CNT100;
   1:  PR[91,1] = PR[90,1] + -38.793;
   1:  PR[91,2] = PR[90,2] + 10.896;
   1:L PR[91] R[100]mm/sec CNT100;
   1:  PR[91,1] = PR[90,1] + -38.989;
   1:  PR[91,2] = PR[90,2] + 10.556;
   1:L PR[91] R[100]mm/sec CNT100;
   1:  PR[91,1] = PR[90,1] + -40.774;
   1:  PR[91,2] = PR[90,2] + 8.007;
   1:L PR[91] R[100]mm/sec CNT100;
   1:  PR[91,1] = PR[90,1] + -41.942;
   1:  PR[91,2] = PR[90,2] + 5.501;
   1:L PR[91] R[100]mm/sec CNT100;
   1:  PR[91,1] = PR[90,1] + -42.010;
   1:  PR[91,2] = PR[90,2] + 5.114;
   1:L PR[91] R[100]mm/sec CNT100;
   1:  PR[91,1] = PR[90,1] + -42.815;
   1:  PR[91,2] = PR[90,2] + 2.108;
   1:L PR[91] R[100]mm/sec CNT100;
   1:  PR[91,1] = PR[90,1] + -43.055;
   1:  PR[91,2] = PR[90,2] + -0.641;
   1:L PR[91] R[100]mm/sec CNT100TB   .50sec,CALL END_PUD;
   1:  PR[92] = PR[91];
   1:  PR[92,3] = PR[92,3] + 20;
   1:J PR[92] 10% FINE;
   1:  PR[91,1] = PR[90,1] + 36.259;
   1:  PR[91,2] = PR[90,2] + 13.219;
   1:  PR[92] = PR[91];
   1:  PR[92,3] = PR[92,3] + 20;
   1:J PR[92] 10% FINE;
   1:L PR[91] R[100]mm/sec CNT100;
   1:  CALL LASER_DRAHT_START;
   1:  PR[91,1] = PR[90,1] + 33.991;
   1:  PR[91,2] = PR[90,2] + 14.806;
   1:L PR[91] R[100]mm/sec CNT100;
   1:  PR[91,1] = PR[90,1] + 33.622;
   1:  PR[91,2] = PR[90,2] + 14.940;
   1:L PR[91] R[100]mm/sec CNT100;
   1:  PR[91,1] = PR[90,1] + 30.804;
   1:  PR[91,2] = PR[90,2] + 16.253;
   1:L PR[91] R[100]mm/sec CNT100;
   1:  PR[91,1] = PR[90,1] + 28.132;
   1:  PR[91,2] = PR[90,2] + 16.968;
   1:L PR[91] R[100]mm/sec CNT100;
   1:  PR[91,1] = PR[90,1] + 27.739;
   1:L PR[91] R[100]mm/sec CNT100;
   1:  PR[91,1] = PR[90,1] + 24.639;
   1:  PR[91,2] = PR[90,2] + 17.238;
   1:L PR[91] R[100]mm/sec CNT100;
   1:  PR[91,1] = PR[90,1] + 21.889;
   1:  PR[91,2] = PR[90,2] + 16.997;
   1:L PR[91] R[100]mm/sec CNT100;
   1:  PR[91,1] = PR[90,1] + 21.520;
   1:  PR[91,2] = PR[90,2] + 16.862;
   1:L PR[91] R[100]mm/sec CNT100;
   1:  PR[91,1] = PR[90,1] + 18.512;
   1:  PR[91,2] = PR[90,2] + 16.055;
   1:L PR[91] R[100]mm/sec CNT100;
   1:  PR[91,1] = PR[90,1] + 15.934;
   1:  PR[91,2] = PR[90,2] + 14.853;
   1:L PR[91] R[100]mm/sec CNT100;
   1:  PR[91,1] = PR[90,1] + 13.524;
   1:  PR[91,2] = PR[90,2] + 13.165;
   1:L PR[91] R[100]mm/sec CNT100;
   1:  PR[91,1] = PR[90,1] + 13.222;
   1:  PR[91,2] = PR[90,2] + 12.912;
   1:L PR[91] R[100]mm/sec CNT100;
   1:  PR[91,1] = PR[90,1] + 11.148;
   1:  PR[91,2] = PR[90,2] + 10.838;
   1:L PR[91] R[100]mm/sec CNT100;
   1:  PR[91,1] = PR[90,1] + 9.460;
   1:  PR[91,2] = PR[90,2] + 8.426;
   1:L PR[91] R[100]mm/sec CNT100;
   1:  PR[91,1] = PR[90,1] + 9.263;
   1:  PR[91,2] = PR[90,2] + 8.085;
   1:L PR[91] R[100]mm/sec CNT100;
   1:  PR[91,1] = PR[90,1] + 8.059;
   1:  PR[91,2] = PR[90,2] + 5.504;
   1:L PR[91] R[100]mm/sec CNT100;
   1:  PR[91,1] = PR[90,1] + 7.991;
   1:  PR[91,2] = PR[90,2] + 5.117;
   1:L PR[91] R[100]mm/sec CNT100;
   1:  PR[91,1] = PR[90,1] + 7.185;
   1:  PR[91,2] = PR[90,2] + 2.107;
   1:L PR[91] R[100]mm/sec CNT100;
   1:  PR[91,1] = PR[90,1] + 6.945;
   1:  PR[91,2] = PR[90,2] + -0.641;
   1:L PR[91] R[100]mm/sec CNT100;
   1:  PR[91,1] = PR[90,1] + 7.013;
   1:  PR[91,2] = PR[90,2] + -1.028;
   1:L PR[91] R[100]mm/sec CNT100;
   1:  PR[91,1] = PR[90,1] + 7.284;
   1:  PR[91,2] = PR[90,2] + -4.126;
   1:L PR[91] R[100]mm/sec CNT100;
   1:  PR[91,1] = PR[90,1] + 8.000;
   1:  PR[91,2] = PR[90,2] + -6.799;
   1:L PR[91] R[100]mm/sec CNT100;
   1:  PR[91,1] = PR[90,1] + 8.196;
   1:  PR[91,2] = PR[90,2] + -7.139;
   1:L PR[91] R[100]mm/sec CNT100;
   1:  PR[91,1] = PR[90,1] + 9.512;
   1:  PR[91,2] = PR[90,2] + -9.960;
   1:L PR[91] R[100]mm/sec CNT100;
   1:  PR[91,1] = PR[90,1] + 11.101;
   1:  PR[91,2] = PR[90,2] + -12.228;
   1:L PR[91] R[100]mm/sec CNT100;
   1:  PR[91,1] = PR[90,1] + 11.401;
   1:  PR[91,2] = PR[90,2] + -12.480;
   1:L PR[91] R[100]mm/sec CNT100;
   1:  PR[91,1] = PR[90,1] + 13.600;
   1:  PR[91,2] = PR[90,2] + -14.678;
   1:L PR[91] R[100]mm/sec CNT100;
   1:  PR[91,1] = PR[90,1] + 15.868;
   1:  PR[91,2] = PR[90,2] + -16.265;
   1:L PR[91] R[100]mm/sec CNT100;
   1:  PR[91,1] = PR[90,1] + 16.237;
   1:  PR[91,2] = PR[90,2] + -16.399;
   1:L PR[91] R[100]mm/sec CNT100;
   1:  PR[91,1] = PR[90,1] + 19.055;
   1:  PR[91,2] = PR[90,2] + -17.712;
   1:L PR[91] R[100]mm/sec CNT100;
   1:  PR[91,1] = PR[90,1] + 21.727;
   1:  PR[91,2] = PR[90,2] + -18.427;
   1:L PR[91] R[100]mm/sec CNT100;
   1:  PR[91,1] = PR[90,1] + 22.120;
   1:L PR[91] R[100]mm/sec CNT100;
   1:  PR[91,1] = PR[90,1] + 25.220;
   1:  PR[91,2] = PR[90,2] + -18.697;
   1:L PR[91] R[100]mm/sec CNT100;
   1:  PR[91,1] = PR[90,1] + 27.970;
   1:  PR[91,2] = PR[90,2] + -18.455;
   1:L PR[91] R[100]mm/sec CNT100;
   1:  PR[91,1] = PR[90,1] + 28.339;
   1:  PR[91,2] = PR[90,2] + -18.321;
   1:L PR[91] R[100]mm/sec CNT100;
   1:  PR[91,1] = PR[90,1] + 31.347;
   1:  PR[91,2] = PR[90,2] + -17.514;
   1:L PR[91] R[100]mm/sec CNT100;
   1:  PR[91,1] = PR[90,1] + 33.925;
   1:  PR[91,2] = PR[90,2] + -16.311;
   1:L PR[91] R[100]mm/sec CNT100;
   1:  PR[91,1] = PR[90,1] + 36.335;
   1:  PR[91,2] = PR[90,2] + -14.624;
   1:L PR[91] R[100]mm/sec CNT100;
   1:  PR[91,1] = PR[90,1] + 36.637;
   1:  PR[91,2] = PR[90,2] + -14.371;
   1:L PR[91] R[100]mm/sec CNT100;
   1:  PR[91,1] = PR[90,1] + 38.710;
   1:  PR[91,2] = PR[90,2] + -12.297;
   1:L PR[91] R[100]mm/sec CNT100;
   1:  PR[91,1] = PR[90,1] + 40.399;
   1:  PR[91,2] = PR[90,2] + -9.885;
   1:L PR[91] R[100]mm/sec CNT100;
   1:  PR[91,1] = PR[90,1] + 40.596;
   1:  PR[91,2] = PR[90,2] + -9.544;
   1:L PR[91] R[100]mm/sec CNT100;
   1:  PR[91,1] = PR[90,1] + 41.799;
   1:  PR[91,2] = PR[90,2] + -6.963;
   1:L PR[91] R[100]mm/sec CNT100;
   1:  PR[91,1] = PR[90,1] + 41.868;
   1:  PR[91,2] = PR[90,2] + -6.576;
   1:L PR[91] R[100]mm/sec CNT100;
   1:  PR[91,1] = PR[90,1] + 42.674;
   1:  PR[91,2] = PR[90,2] + -3.565;
   1:L PR[91] R[100]mm/sec CNT100;
   1:  PR[91,1] = PR[90,1] + 42.914;
   1:  PR[91,2] = PR[90,2] + -0.818;
   1:L PR[91] R[100]mm/sec CNT100;
   1:  PR[91,1] = PR[90,1] + 42.846;
   1:  PR[91,2] = PR[90,2] + -0.430;
   1:L PR[91] R[100]mm/sec CNT100;
   1:  PR[91,1] = PR[90,1] + 42.575;
   1:  PR[91,2] = PR[90,2] + 2.667;
   1:L PR[91] R[100]mm/sec CNT100;
   1:  PR[91,1] = PR[90,1] + 41.859;
   1:  PR[91,2] = PR[90,2] + 5.341;
   1:L PR[91] R[100]mm/sec CNT100;
   1:  PR[91,1] = PR[90,1] + 41.663;
   1:  PR[91,2] = PR[90,2] + 5.680;
   1:L PR[91] R[100]mm/sec CNT100;
   1:  PR[91,1] = PR[90,1] + 40.347;
   1:  PR[91,2] = PR[90,2] + 8.501;
   1:L PR[91] R[100]mm/sec CNT100;
   1:  PR[91,1] = PR[90,1] + 38.758;
   1:  PR[91,2] = PR[90,2] + 10.769;
   1:L PR[91] R[100]mm/sec CNT100;
   1:  PR[91,1] = PR[90,1] + 38.457;
   1:  PR[91,2] = PR[90,2] + 11.022;
   1:L PR[91] R[100]mm/sec CNT100;
   1:  PR[91,1] = PR[90,1] + 36.259;
   1:  PR[91,2] = PR[90,2] + 13.219;
   1:L PR[91] R[100]mm/sec CNT100TB   .50sec,CALL END_PUD;
   1:  PR[92] = PR[91];
   1:  PR[92,3] = PR[92,3] + 20;
   1:J PR[92] 10% FINE;
   1:  PR[91,1] = PR[90,1] + 59.263;
   1:  PR[91,2] = PR[90,2] + -9.544;
   1:  PR[92] = PR[91];
   1:  PR[92,3] = PR[92,3] + 20;
   1:J PR[92] 10% FINE;
   1:L PR[91] R[100]mm/sec CNT100;
   1:  CALL LASER_DRAHT_START;
   1:  PR[91,1] = PR[90,1] + 59.460;
   1:  PR[91,2] = PR[90,2] + -9.885;
   1:L PR[91] R[100]mm/sec CNT100;
   1:  PR[91,1] = PR[90,1] + 61.098;
   1:  PR[91,2] = PR[90,2] + -12.225;
   1:L PR[91] R[100]mm/sec CNT100;
   1:  PR[91,1] = PR[90,1] + 61.398;
   1:  PR[91,2] = PR[90,2] + -12.477;
   1:L PR[91] R[100]mm/sec CNT100;
   1:  PR[91,1] = PR[90,1] + 63.596;
   1:  PR[91,2] = PR[90,2] + -14.674;
   1:L PR[91] R[100]mm/sec CNT100;
   1:  PR[91,1] = PR[90,1] + 65.861;
   1:  PR[91,2] = PR[90,2] + -16.261;
   1:L PR[91] R[100]mm/sec CNT100;
   1:  PR[91,1] = PR[90,1] + 66.230;
   1:  PR[91,2] = PR[90,2] + -16.395;
   1:L PR[91] R[100]mm/sec CNT100;
   1:  PR[91,1] = PR[90,1] + 69.046;
   1:  PR[91,2] = PR[90,2] + -17.709;
   1:L PR[91] R[100]mm/sec CNT100;
   1:  PR[91,1] = PR[90,1] + 71.801;
   1:  PR[91,2] = PR[90,2] + -18.448;
   1:L PR[91] R[100]mm/sec CNT100;
   1:  PR[91,1] = PR[90,1] + 74.726;
   1:  PR[91,2] = PR[90,2] + -18.704;
   1:L PR[91] R[100]mm/sec CNT100;
   1:  PR[91,1] = PR[90,1] + 75.120;
   1:L PR[91] R[100]mm/sec CNT100;
   1:  PR[91,1] = PR[90,1] + 78.047;
   1:  PR[91,2] = PR[90,2] + -18.450;
   1:L PR[91] R[100]mm/sec CNT100;
   1:  PR[91,1] = PR[90,1] + 80.888;
   1:  PR[91,2] = PR[90,2] + -17.689;
   1:L PR[91] R[100]mm/sec CNT100;
   1:  PR[91,1] = PR[90,1] + 81.258;
   1:  PR[91,2] = PR[90,2] + -17.555;
   1:L PR[91] R[100]mm/sec CNT100;
   1:  PR[91,1] = PR[90,1] + 83.919;
   1:  PR[91,2] = PR[90,2] + -16.315;
   1:L PR[91] R[100]mm/sec CNT100;
   1:  PR[91,1] = PR[90,1] + 86.330;
   1:  PR[91,2] = PR[90,2] + -14.628;
   1:L PR[91] R[100]mm/sec CNT100;
   1:  PR[91,1] = PR[90,1] + 86.632;
   1:  PR[91,2] = PR[90,2] + -14.375;
   1:L PR[91] R[100]mm/sec CNT100;
   1:  PR[91,1] = PR[90,1] + 88.708;
   1:  PR[91,2] = PR[90,2] + -12.300;
   1:L PR[91] R[100]mm/sec CNT100;
   1:  PR[91,1] = PR[90,1] + 90.398;
   1:  PR[91,2] = PR[90,2] + -9.888;
   1:L PR[91] R[100]mm/sec CNT100;
   1:  PR[91,1] = PR[90,1] + 90.594;
   1:  PR[91,2] = PR[90,2] + -9.547;
   1:L PR[91] R[100]mm/sec CNT100;
   1:  PR[91,1] = PR[90,1] + 91.836;
   1:  PR[91,2] = PR[90,2] + -6.885;
   1:L PR[91] R[100]mm/sec CNT100;
   1:  PR[91,1] = PR[90,1] + 92.598;
   1:  PR[91,2] = PR[90,2] + -4.041;
   1:L PR[91] R[100]mm/sec CNT100;
   1:  PR[91,1] = PR[90,1] + 92.666;
   1:  PR[91,2] = PR[90,2] + -3.653;
   1:L PR[91] R[100]mm/sec CNT100;
   1:  PR[91,1] = PR[90,1] + 92.914;
   1:  PR[91,2] = PR[90,2] + -0.818;
   1:L PR[91] R[100]mm/sec CNT100;
   1:  PR[91,1] = PR[90,1] + 92.846;
   1:  PR[91,2] = PR[90,2] + -0.430;
   1:L PR[91] R[100]mm/sec CNT100;
   1:  PR[91,1] = PR[90,1] + 92.575;
   1:  PR[91,2] = PR[90,2] + 2.667;
   1:L PR[91] R[100]mm/sec CNT100;
   1:  PR[91,1] = PR[90,1] + 91.837;
   1:  PR[91,2] = PR[90,2] + 5.424;
   1:L PR[91] R[100]mm/sec CNT100;
   1:  PR[91,1] = PR[90,1] + 90.596;
   1:  PR[91,2] = PR[90,2] + 8.085;
   1:L PR[91] R[100]mm/sec CNT100;
   1:  PR[91,1] = PR[90,1] + 90.399;
   1:  PR[91,2] = PR[90,2] + 8.426;
   1:L PR[91] R[100]mm/sec CNT100;
   1:  PR[91,1] = PR[90,1] + 88.761;
   1:  PR[91,2] = PR[90,2] + 10.766;
   1:L PR[91] R[100]mm/sec CNT100;
   1:  PR[91,1] = PR[90,1] + 88.460;
   1:  PR[91,2] = PR[90,2] + 11.018;
   1:L PR[91] R[100]mm/sec CNT100;
   1:  PR[91,1] = PR[90,1] + 86.263;
   1:  PR[91,2] = PR[90,2] + 13.215;
   1:L PR[91] R[100]mm/sec CNT100;
   1:  PR[91,1] = PR[90,1] + 83.998;
   1:  PR[91,2] = PR[90,2] + 14.802;
   1:L PR[91] R[100]mm/sec CNT100;
   1:  PR[91,1] = PR[90,1] + 83.628;
   1:  PR[91,2] = PR[90,2] + 14.936;
   1:L PR[91] R[100]mm/sec CNT100;
   1:  PR[91,1] = PR[90,1] + 80.812;
   1:  PR[91,2] = PR[90,2] + 16.250;
   1:L PR[91] R[100]mm/sec CNT100;
   1:  PR[91,1] = PR[90,1] + 78.058;
   1:  PR[91,2] = PR[90,2] + 16.989;
   1:L PR[91] R[100]mm/sec CNT100;
   1:  PR[91,1] = PR[90,1] + 75.133;
   1:  PR[91,2] = PR[90,2] + 17.246;
   1:L PR[91] R[100]mm/sec CNT100;
   1:  PR[91,1] = PR[90,1] + 74.739;
   1:L PR[91] R[100]mm/sec CNT100;
   1:  PR[91,1] = PR[90,1] + 71.812;
   1:  PR[91,2] = PR[90,2] + 16.991;
   1:L PR[91] R[100]mm/sec CNT100;
   1:  PR[91,1] = PR[90,1] + 68.971;
   1:  PR[91,2] = PR[90,2] + 16.231;
   1:L PR[91] R[100]mm/sec CNT100;
   1:  PR[91,1] = PR[90,1] + 68.601;
   1:  PR[91,2] = PR[90,2] + 16.096;
   1:L PR[91] R[100]mm/sec CNT100;
   1:  PR[91,1] = PR[90,1] + 65.940;
   1:  PR[91,2] = PR[90,2] + 14.856;
   1:L PR[91] R[100]mm/sec CNT100;
   1:  PR[91,1] = PR[90,1] + 63.529;
   1:  PR[91,2] = PR[90,2] + 13.169;
   1:L PR[91] R[100]mm/sec CNT100;
   1:  PR[91,1] = PR[90,1] + 63.227;
   1:  PR[91,2] = PR[90,2] + 12.916;
   1:L PR[91] R[100]mm/sec CNT100;
   1:  PR[91,1] = PR[90,1] + 61.151;
   1:  PR[91,2] = PR[90,2] + 10.841;
   1:L PR[91] R[100]mm/sec CNT100;
   1:  PR[91,1] = PR[90,1] + 59.461;
   1:  PR[91,2] = PR[90,2] + 8.429;
   1:L PR[91] R[100]mm/sec CNT100;
   1:  PR[91,1] = PR[90,1] + 59.264;
   1:  PR[91,2] = PR[90,2] + 8.088;
   1:L PR[91] R[100]mm/sec CNT100;
   1:  PR[91,1] = PR[90,1] + 58.023;
   1:  PR[91,2] = PR[90,2] + 5.426;
   1:L PR[91] R[100]mm/sec CNT100;
   1:  PR[91,1] = PR[90,1] + 57.261;
   1:  PR[91,2] = PR[90,2] + 2.582;
   1:L PR[91] R[100]mm/sec CNT100;
   1:  PR[91,1] = PR[90,1] + 57.192;
   1:  PR[91,2] = PR[90,2] + 2.194;
   1:L PR[91] R[100]mm/sec CNT100;
   1:  PR[91,1] = PR[90,1] + 56.945;
   1:  PR[91,2] = PR[90,2] + -0.641;
   1:L PR[91] R[100]mm/sec CNT100;
   1:  PR[91,1] = PR[90,1] + 57.013;
   1:  PR[91,2] = PR[90,2] + -1.028;
   1:L PR[91] R[100]mm/sec CNT100;
   1:  PR[91,1] = PR[90,1] + 57.284;
   1:  PR[91,2] = PR[90,2] + -4.126;
   1:L PR[91] R[100]mm/sec CNT100;
   1:  PR[91,1] = PR[90,1] + 58.022;
   1:  PR[91,2] = PR[90,2] + -6.883;
   1:L PR[91] R[100]mm/sec CNT100;
   1:  PR[91,1] = PR[90,1] + 59.263;
   1:  PR[91,2] = PR[90,2] + -9.544;
   1:L PR[91] R[100]mm/sec CNT100TB   .50sec,CALL END_PUD;
   1:  PR[92] = PR[91];
   1:  PR[92,3] = PR[92,3] + 20;
   1:J PR[92] 10% FINE;
   1:  PR[91] = PR[90];
   1:  PR[91,1] = PR[90,1] + 38.671;
   1:  PR[91,2] = PR[90,2] + -12.369;
   1:  PR[91,3] = PR[90,3] + 9.295;
   1:  PR[92] = PR[91];
   1:  PR[92,3] = PR[92,3] + 20;
   1:J PR[92] 10% FINE;
   1:L PR[91] R[100]mm/sec CNT100;
   1:  CALL LASER_DRAHT_START;
   1:  PR[91,1] = PR[90,1] + 40.525;
   1:  PR[91,2] = PR[90,2] + -9.736;
   1:L PR[91] R[100]mm/sec CNT100;
   1:  PR[91,1] = PR[90,1] + 41.874;
   1:  PR[91,2] = PR[90,2] + -6.821;
   1:L PR[91] R[100]mm/sec CNT100;
   1:  PR[91,1] = PR[90,1] + 42.649;
   1:  PR[91,2] = PR[90,2] + -3.927;
   1:L PR[91] R[100]mm/sec CNT100;
   1:  PR[91,1] = PR[90,1] + 42.934;
   1:  PR[91,2] = PR[90,2] + -0.729;
   1:L PR[91] R[100]mm/sec CNT100;
   1:  PR[91,1] = PR[90,1] + 42.649;
   1:  PR[91,2] = PR[90,2] + 2.469;
   1:L PR[91] R[100]mm/sec CNT100;
   1:  PR[91,1] = PR[90,1] + 41.862;
   1:  PR[91,2] = PR[90,2] + 5.404;
   1:L PR[91] R[100]mm/sec CNT100;
   1:  PR[91,1] = PR[90,1] + 41.841;
   1:  PR[91,2] = PR[90,2] + 5.456;
   1:L PR[91] R[100]mm/sec CNT100;
   1:  PR[91,1] = PR[90,1] + 40.524;
   1:  PR[91,2] = PR[90,2] + 8.280;
   1:L PR[91] R[100]mm/sec CNT100;
   1:  PR[91,1] = PR[90,1] + 38.730;
   1:  PR[91,2] = PR[90,2] + 10.841;
   1:L PR[91] R[100]mm/sec CNT100;
   1:  PR[91,1] = PR[90,1] + 38.696;
   1:  PR[91,2] = PR[90,2] + 10.886;
   1:L PR[91] R[100]mm/sec CNT100;
   1:  PR[91,1] = PR[90,1] + 36.555;
   1:  PR[91,2] = PR[90,2] + 13.025;
   1:L PR[91] R[100]mm/sec CNT100;
   1:  PR[91,1] = PR[90,1] + 33.922;
   1:  PR[91,2] = PR[90,2] + 14.879;
   1:L PR[91] R[100]mm/sec CNT100;
   1:  PR[91,1] = PR[90,1] + 31.006;
   1:  PR[91,2] = PR[90,2] + 16.228;
   1:L PR[91] R[100]mm/sec CNT100;
   1:  PR[91,1] = PR[90,1] + 28.074;
   1:  PR[91,2] = PR[90,2] + 17.012;
   1:L PR[91] R[100]mm/sec CNT100;
   1:  PR[91,1] = PR[90,1] + 28.012;
   1:  PR[91,2] = PR[90,2] + 17.021;
   1:L PR[91] R[100]mm/sec CNT100;
   1:  PR[91,1] = PR[90,1] + 24.916;
   1:  PR[91,2] = PR[90,2] + 17.290;
   1:L PR[91] R[100]mm/sec CNT100;
   1:  PR[91,1] = PR[90,1] + 21.710;
   1:  PR[91,2] = PR[90,2] + 17.000;
   1:L PR[91] R[100]mm/sec CNT100;
   1:  PR[91,1] = PR[90,1] + 18.829;
   1:  PR[91,2] = PR[90,2] + 16.227;
   1:L PR[91] R[100]mm/sec CNT100;
   1:  PR[91,1] = PR[90,1] + 15.934;
   1:  PR[91,2] = PR[90,2] + 14.876;
   1:L PR[91] R[100]mm/sec CNT100;
   1:  PR[91,1] = PR[90,1] + 15.875;
   1:  PR[91,2] = PR[90,2] + 14.852;
   1:L PR[91] R[100]mm/sec CNT100;
   1:  PR[91,1] = PR[90,1] + 13.275;
   1:  PR[91,2] = PR[90,2] + 13.020;
   1:L PR[91] R[100]mm/sec CNT100;
   1:  PR[91,1] = PR[90,1] + 11.141;
   1:  PR[91,2] = PR[90,2] + 10.886;
   1:L PR[91] R[100]mm/sec CNT100;
   1:  PR[91,1] = PR[90,1] + 11.096;
   1:  PR[91,2] = PR[90,2] + 10.828;
   1:L PR[91] R[100]mm/sec CNT100;
   1:  PR[91,1] = PR[90,1] + 9.313;
   1:  PR[91,2] = PR[90,2] + 8.281;
   1:L PR[91] R[100]mm/sec CNT100;
   1:  PR[91,1] = PR[90,1] + 7.961;
   1:  PR[91,2] = PR[90,2] + 5.358;
   1:L PR[91] R[100]mm/sec CNT100;
   1:  PR[91,1] = PR[90,1] + 7.189;
   1:  PR[91,2] = PR[90,2] + 2.474;
   1:L PR[91] R[100]mm/sec CNT100;
   1:  PR[91,1] = PR[90,1] + 6.899;
   1:  PR[91,2] = PR[90,2] + -0.733;
   1:L PR[91] R[100]mm/sec CNT100;
   1:  PR[91,1] = PR[90,1] + 7.168;
   1:  PR[91,2] = PR[90,2] + -3.819;
   1:L PR[91] R[100]mm/sec CNT100;
   1:  PR[91,1] = PR[90,1] + 7.178;
   1:  PR[91,2] = PR[90,2] + -3.894;
   1:L PR[91] R[100]mm/sec CNT100;
   1:  PR[91,1] = PR[90,1] + 7.972;
   1:  PR[91,2] = PR[90,2] + -6.857;
   1:L PR[91] R[100]mm/sec CNT100;
   1:  PR[91,1] = PR[90,1] + 8.000;
   1:  PR[91,2] = PR[90,2] + -6.925;
   1:L PR[91] R[100]mm/sec CNT100;
   1:  PR[91,1] = PR[90,1] + 9.313;
   1:  PR[91,2] = PR[90,2] + -9.740;
   1:L PR[91] R[100]mm/sec CNT100;
   1:  PR[91,1] = PR[90,1] + 11.099;
   1:  PR[91,2] = PR[90,2] + -12.290;
   1:L PR[91] R[100]mm/sec CNT100;
   1:  PR[91,1] = PR[90,1] + 11.144;
   1:  PR[91,2] = PR[90,2] + -12.348;
   1:L PR[91] R[100]mm/sec CNT100;
   1:  PR[91,1] = PR[90,1] + 13.280;
   1:  PR[91,2] = PR[90,2] + -14.483;
   1:L PR[91] R[100]mm/sec CNT100;
   1:  PR[91,1] = PR[90,1] + 15.919;
   1:  PR[91,2] = PR[90,2] + -16.341;
   1:L PR[91] R[100]mm/sec CNT100;
   1:  PR[91,1] = PR[90,1] + 18.731;
   1:  PR[91,2] = PR[90,2] + -17.651;
   1:L PR[91] R[100]mm/sec CNT100;
   1:  PR[91,1] = PR[90,1] + 18.794;
   1:  PR[91,2] = PR[90,2] + -17.677;
   1:L PR[91] R[100]mm/sec CNT100;
   1:  PR[91,1] = PR[90,1] + 21.722;
   1:  PR[91,2] = PR[90,2] + -18.460;
   1:L PR[91] R[100]mm/sec CNT100;
   1:  PR[91,1] = PR[90,1] + 24.929;
   1:  PR[91,2] = PR[90,2] + -18.749;
   1:L PR[91] R[100]mm/sec CNT100;
   1:  PR[91,1] = PR[90,1] + 28.024;
   1:  PR[91,2] = PR[90,2] + -18.477;
   1:L PR[91] R[100]mm/sec CNT100;
   1:  PR[91,1] = PR[90,1] + 28.086;
   1:  PR[91,2] = PR[90,2] + -18.469;
   1:L PR[91] R[100]mm/sec CNT100;
   1:  PR[91,1] = PR[90,1] + 31.015;
   1:  PR[91,2] = PR[90,2] + -17.683;
   1:L PR[91] R[100]mm/sec CNT100;
   1:  PR[91,1] = PR[90,1] + 33.931;
   1:  PR[91,2] = PR[90,2] + -16.333;
   1:L PR[91] R[100]mm/sec CNT100;
   1:  PR[91,1] = PR[90,1] + 36.483;
   1:  PR[91,2] = PR[90,2] + -14.546;
   1:L PR[91] R[100]mm/sec CNT100;
   1:  PR[91,1] = PR[90,1] + 36.530;
   1:  PR[91,2] = PR[90,2] + -14.510;
   1:L PR[91] R[100]mm/sec CNT100;
   1:  PR[91,1] = PR[90,1] + 38.671;
   1:  PR[91,2] = PR[90,2] + -12.369;
   1:L PR[91] R[100]mm/sec CNT100TB   .50sec,CALL END_PUD;
   1:  PR[92] = PR[91];
   1:  PR[92,3] = PR[92,3] + 20;
   1:J PR[92] 10% FINE;
   1:  PR[91,1] = PR[90,1] + 63.346;
   1:  PR[91,2] = PR[90,2] + 13.103;
   1:  PR[92] = PR[91];
   1:  PR[92,3] = PR[92,3] + 20;
   1:J PR[92] 10% FINE;
   1:L PR[91] R[100]mm/sec CNT100;
   1:  CALL LASER_DRAHT_START;
   1:  PR[91,1] = PR[90,1] + 61.062;
   1:  PR[91,2] = PR[90,2] + 10.822;
   1:L PR[91] R[100]mm/sec CNT100;
   1:  PR[91,1] = PR[90,1] + 59.371;
   1:  PR[91,2] = PR[90,2] + 8.408;
   1:L PR[91] R[100]mm/sec CNT100;
   1:  PR[91,1] = PR[90,1] + 59.236;
   1:  PR[91,2] = PR[90,2] + 8.195;
   1:L PR[91] R[100]mm/sec CNT100;
   1:  PR[91,1] = PR[90,1] + 58.000;
   1:  PR[91,2] = PR[90,2] + 5.546;
   1:L PR[91] R[100]mm/sec CNT100;
   1:  PR[91,1] = PR[90,1] + 57.911;
   1:  PR[91,2] = PR[90,2] + 5.291;
   1:L PR[91] R[100]mm/sec CNT100;
   1:  PR[91,1] = PR[90,1] + 57.161;
   1:  PR[91,2] = PR[90,2] + 2.492;
   1:L PR[91] R[100]mm/sec CNT100;
   1:  PR[91,1] = PR[90,1] + 56.869;
   1:  PR[91,2] = PR[90,2] + -0.729;
   1:L PR[91] R[100]mm/sec CNT100;
   1:  PR[91,1] = PR[90,1] + 57.161;
   1:  PR[91,2] = PR[90,2] + -3.950;
   1:L PR[91] R[100]mm/sec CNT100;
   1:  PR[91,1] = PR[90,1] + 57.910;
   1:  PR[91,2] = PR[90,2] + -6.748;
   1:L PR[91] R[100]mm/sec CNT100;
   1:  PR[91,1] = PR[90,1] + 58.000;
   1:  PR[91,2] = PR[90,2] + -7.003;
   1:L PR[91] R[100]mm/sec CNT100;
   1:  PR[91,1] = PR[90,1] + 59.234;
   1:  PR[91,2] = PR[90,2] + -9.651;
   1:L PR[91] R[100]mm/sec CNT100;
   1:  PR[91,1] = PR[90,1] + 59.369;
   1:  PR[91,2] = PR[90,2] + -9.864;
   1:L PR[91] R[100]mm/sec CNT100;
   1:  PR[91,1] = PR[90,1] + 61.059;
   1:  PR[91,2] = PR[90,2] + -12.278;
   1:L PR[91] R[100]mm/sec CNT100;
   1:  PR[91,1] = PR[90,1] + 63.165;
   1:  PR[91,2] = PR[90,2] + -14.384;
   1:L PR[91] R[100]mm/sec CNT100;
   1:  PR[91,1] = PR[90,1] + 63.338;
   1:  PR[91,2] = PR[90,2] + -14.556;
   1:L PR[91] R[100]mm/sec CNT100;
   1:  PR[91,1] = PR[90,1] + 65.762;
   1:  PR[91,2] = PR[90,2] + -16.253;
   1:L PR[91] R[100]mm/sec CNT100;
   1:  PR[91,1] = PR[90,1] + 65.946;
   1:  PR[91,2] = PR[90,2] + -16.367;
   1:L PR[91] R[100]mm/sec CNT100;
   1:  PR[91,1] = PR[90,1] + 68.635;
   1:  PR[91,2] = PR[90,2] + -17.622;
   1:L PR[91] R[100]mm/sec CNT100;
   1:  PR[91,1] = PR[90,1] + 68.812;
   1:  PR[91,2] = PR[90,2] + -17.683;
   1:L PR[91] R[100]mm/sec CNT100;
   1:  PR[91,1] = PR[90,1] + 71.684;
   1:  PR[91,2] = PR[90,2] + -18.453;
   1:L PR[91] R[100]mm/sec CNT100;
   1:  PR[91,1] = PR[90,1] + 74.884;
   1:  PR[91,2] = PR[90,2] + -18.740;
   1:L PR[91] R[100]mm/sec CNT100;
   1:  PR[91,1] = PR[90,1] + 78.077;
   1:  PR[91,2] = PR[90,2] + -18.454;
   1:L PR[91] R[100]mm/sec CNT100;
   1:  PR[91,1] = PR[90,1] + 80.974;
   1:  PR[91,2] = PR[90,2] + -17.678;
   1:L PR[91] R[100]mm/sec CNT100;
   1:  PR[91,1] = PR[90,1] + 81.096;
   1:  PR[91,2] = PR[90,2] + -17.635;
   1:L PR[91] R[100]mm/sec CNT100;
   1:  PR[91,1] = PR[90,1] + 83.843;
   1:  PR[91,2] = PR[90,2] + -16.355;
   1:L PR[91] R[100]mm/sec CNT100;
   1:  PR[91,1] = PR[90,1] + 83.938;
   1:  PR[91,2] = PR[90,2] + -16.296;
   1:L PR[91] R[100]mm/sec CNT100;
   1:  PR[91,1] = PR[90,1] + 86.439;
   1:  PR[91,2] = PR[90,2] + -14.546;
   1:L PR[91] R[100]mm/sec CNT100;
   1:  PR[91,1] = PR[90,1] + 88.699;
   1:  PR[91,2] = PR[90,2] + -12.286;
   1:L PR[91] R[100]mm/sec CNT100;
   1:  PR[91,1] = PR[90,1] + 90.453;
   1:  PR[91,2] = PR[90,2] + -9.782;
   1:L PR[91] R[100]mm/sec CNT100;
   1:  PR[91,1] = PR[90,1] + 90.503;
   1:  PR[91,2] = PR[90,2] + -9.701;
   1:L PR[91] R[100]mm/sec CNT100;
   1:  PR[91,1] = PR[90,1] + 91.795;
   1:  PR[91,2] = PR[90,2] + -6.931;
   1:L PR[91] R[100]mm/sec CNT100;
   1:  PR[91,1] = PR[90,1] + 91.824;
   1:  PR[91,2] = PR[90,2] + -6.848;
   1:L PR[91] R[100]mm/sec CNT100;
   1:  PR[91,1] = PR[90,1] + 92.612;
   1:  PR[91,2] = PR[90,2] + -3.907;
   1:L PR[91] R[100]mm/sec CNT100;
   1:  PR[91,1] = PR[90,1] + 92.895;
   1:  PR[91,2] = PR[90,2] + -0.729;
   1:L PR[91] R[100]mm/sec CNT100;
   1:  PR[91,1] = PR[90,1] + 92.612;
   1:  PR[91,2] = PR[90,2] + 2.448;
   1:L PR[91] R[100]mm/sec CNT100;
   1:  PR[91,1] = PR[90,1] + 91.825;
   1:  PR[91,2] = PR[90,2] + 5.387;
   1:L PR[91] R[100]mm/sec CNT100;
   1:  PR[91,1] = PR[90,1] + 91.796;
   1:  PR[91,2] = PR[90,2] + 5.470;
   1:L PR[91] R[100]mm/sec CNT100;
   1:  PR[91,1] = PR[90,1] + 90.505;
   1:  PR[91,2] = PR[90,2] + 8.239;
   1:L PR[91] R[100]mm/sec CNT100;
   1:  PR[91,1] = PR[90,1] + 90.455;
   1:  PR[91,2] = PR[90,2] + 8.320;
   1:L PR[91] R[100]mm/sec CNT100;
   1:  PR[91,1] = PR[90,1] + 88.702;
   1:  PR[91,2] = PR[90,2] + 10.824;
   1:L PR[91] R[100]mm/sec CNT100;
   1:  PR[91,1] = PR[90,1] + 86.443;
   1:  PR[91,2] = PR[90,2] + 13.083;
   1:L PR[91] R[100]mm/sec CNT100;
   1:  PR[91,1] = PR[90,1] + 83.945;
   1:  PR[91,2] = PR[90,2] + 14.833;
   1:L PR[91] R[100]mm/sec CNT100;
   1:  PR[91,1] = PR[90,1] + 83.850;
   1:  PR[91,2] = PR[90,2] + 14.893;
   1:L PR[91] R[100]mm/sec CNT100;
   1:  PR[91,1] = PR[90,1] + 81.106;
   1:  PR[91,2] = PR[90,2] + 16.173;
   1:L PR[91] R[100]mm/sec CNT100;
   1:  PR[91,1] = PR[90,1] + 80.983;
   1:  PR[91,2] = PR[90,2] + 16.216;
   1:L PR[91] R[100]mm/sec CNT100;
   1:  PR[91,1] = PR[90,1] + 78.088;
   1:  PR[91,2] = PR[90,2] + 16.993;
   1:L PR[91] R[100]mm/sec CNT100;
   1:  PR[91,1] = PR[90,1] + 74.897;
   1:  PR[91,2] = PR[90,2] + 17.282;
   1:L PR[91] R[100]mm/sec CNT100;
   1:  PR[91,1] = PR[90,1] + 71.695;
   1:  PR[91,2] = PR[90,2] + 16.996;
   1:L PR[91] R[100]mm/sec CNT100;
   1:  PR[91,1] = PR[90,1] + 68.822;
   1:  PR[91,2] = PR[90,2] + 16.228;
   1:L PR[91] R[100]mm/sec CNT100;
   1:  PR[91,1] = PR[90,1] + 68.644;
   1:  PR[91,2] = PR[90,2] + 16.166;
   1:L PR[91] R[100]mm/sec CNT100;
   1:  PR[91,1] = PR[90,1] + 65.952;
   1:  PR[91,2] = PR[90,2] + 14.912;
   1:L PR[91] R[100]mm/sec CNT100;
   1:  PR[91,1] = PR[90,1] + 65.769;
   1:  PR[91,2] = PR[90,2] + 14.798;
   1:L PR[91] R[100]mm/sec CNT100;
   1:  PR[91,1] = PR[90,1] + 63.346;
   1:  PR[91,2] = PR[90,2] + 13.103;
   1:L PR[91] R[100]mm/sec CNT100TB   .50sec,CALL END_PUD;
   1:  PR[92] = PR[91];
   1:  PR[92,3] = PR[92,3] + 20;
   1:J PR[92] 10% FINE;
   1:  PR[91,1] = PR[90,1] + -38.849;
   1:  PR[91,2] = PR[90,2] + 10.823;
   1:  PR[92] = PR[91];
   1:  PR[92,3] = PR[92,3] + 20;
   1:J PR[92] 10% FINE;
   1:L PR[91] R[100]mm/sec CNT100;
   1:  CALL LASER_DRAHT_START;
   1:  PR[91,1] = PR[90,1] + -40.623;
   1:  PR[91,2] = PR[90,2] + 8.289;
   1:L PR[91] R[100]mm/sec CNT100;
   1:  PR[91,1] = PR[90,1] + -40.644;
   1:  PR[91,2] = PR[90,2] + 8.256;
   1:L PR[91] R[100]mm/sec CNT100;
   1:  PR[91,1] = PR[90,1] + -41.954;
   1:  PR[91,2] = PR[90,2] + 5.445;
   1:L PR[91] R[100]mm/sec CNT100;
   1:  PR[91,1] = PR[90,1] + -41.965;
   1:  PR[91,2] = PR[90,2] + 5.411;
   1:L PR[91] R[100]mm/sec CNT100;
   1:  PR[91,1] = PR[90,1] + -42.761;
   1:  PR[91,2] = PR[90,2] + 2.438;
   1:L PR[91] R[100]mm/sec CNT100;
   1:  PR[91,1] = PR[90,1] + -43.043;
   1:  PR[91,2] = PR[90,2] + -0.731;
   1:L PR[91] R[100]mm/sec CNT100;
   1:  PR[91,1] = PR[90,1] + -42.772;
   1:  PR[91,2] = PR[90,2] + -3.840;
   1:L PR[91] R[100]mm/sec CNT100;
   1:  PR[91,1] = PR[90,1] + -42.768;
   1:  PR[91,2] = PR[90,2] + -3.873;
   1:L PR[91] R[100]mm/sec CNT100;
   1:  PR[91,1] = PR[90,1] + -41.966;
   1:  PR[91,2] = PR[90,2] + -6.869;
   1:L PR[91] R[100]mm/sec CNT100;
   1:  PR[91,1] = PR[90,1] + -41.954;
   1:  PR[91,2] = PR[90,2] + -6.902;
   1:L PR[91] R[100]mm/sec CNT100;
   1:  PR[91,1] = PR[90,1] + -40.644;
   1:  PR[91,2] = PR[90,2] + -9.713;
   1:L PR[91] R[100]mm/sec CNT100;
   1:  PR[91,1] = PR[90,1] + -40.623;
   1:  PR[91,2] = PR[90,2] + -9.746;
   1:L PR[91] R[100]mm/sec CNT100;
   1:  PR[91,1] = PR[90,1] + -38.850;
   1:  PR[91,2] = PR[90,2] + -12.281;
   1:L PR[91] R[100]mm/sec CNT100;
   1:  PR[91,1] = PR[90,1] + -36.596;
   1:  PR[91,2] = PR[90,2] + -14.536;
   1:L PR[91] R[100]mm/sec CNT100;
   1:  PR[91,1] = PR[90,1] + -34.063;
   1:  PR[91,2] = PR[90,2] + -16.310;
   1:L PR[91] R[100]mm/sec CNT100;
   1:  PR[91,1] = PR[90,1] + -34.023;
   1:  PR[91,2] = PR[90,2] + -16.336;
   1:L PR[91] R[100]mm/sec CNT100;
   1:  PR[91,1] = PR[90,1] + -31.223;
   1:  PR[91,2] = PR[90,2] + -17.642;
   1:L PR[91] R[100]mm/sec CNT100;
   1:  PR[91,1] = PR[90,1] + -31.170;
   1:  PR[91,2] = PR[90,2] + -17.661;
   1:L PR[91] R[100]mm/sec CNT100;
   1:  PR[91,1] = PR[90,1] + -28.218;
   1:  PR[91,2] = PR[90,2] + -18.452;
   1:L PR[91] R[100]mm/sec CNT100;
   1:  PR[91,1] = PR[90,1] + -25.039;
   1:  PR[91,2] = PR[90,2] + -18.737;
   1:L PR[91] R[100]mm/sec CNT100;
   1:  PR[91,1] = PR[90,1] + -21.857;
   1:  PR[91,2] = PR[90,2] + -18.453;
   1:L PR[91] R[100]mm/sec CNT100;
   1:  PR[91,1] = PR[90,1] + -18.913;
   1:  PR[91,2] = PR[90,2] + -17.664;
   1:L PR[91] R[100]mm/sec CNT100;
   1:  PR[91,1] = PR[90,1] + -18.836;
   1:  PR[91,2] = PR[90,2] + -17.638;
   1:L PR[91] R[100]mm/sec CNT100;
   1:  PR[91,1] = PR[90,1] + -16.061;
   1:  PR[91,2] = PR[90,2] + -16.343;
   1:L PR[91] R[100]mm/sec CNT100;
   1:  PR[91,1] = PR[90,1] + -15.982;
   1:  PR[91,2] = PR[90,2] + -16.294;
   1:L PR[91] R[100]mm/sec CNT100;
   1:  PR[91,1] = PR[90,1] + -13.484;
   1:  PR[91,2] = PR[90,2] + -14.545;
   1:L PR[91] R[100]mm/sec CNT100;
   1:  PR[91,1] = PR[90,1] + -11.220;
   1:  PR[91,2] = PR[90,2] + -12.280;
   1:L PR[91] R[100]mm/sec CNT100;
   1:  PR[91,1] = PR[90,1] + -9.472;
   1:  PR[91,2] = PR[90,2] + -9.784;
   1:L PR[91] R[100]mm/sec CNT100;
   1:  PR[91,1] = PR[90,1] + -9.415;
   1:  PR[91,2] = PR[90,2] + -9.693;
   1:L PR[91] R[100]mm/sec CNT100;
   1:  PR[91,1] = PR[90,1] + -8.129;
   1:  PR[91,2] = PR[90,2] + -6.935;
   1:L PR[91] R[100]mm/sec CNT100;
   1:  PR[91,1] = PR[90,1] + -8.092;
   1:  PR[91,2] = PR[90,2] + -6.828;
   1:L PR[91] R[100]mm/sec CNT100;
   1:  PR[91,1] = PR[90,1] + -7.312;
   1:  PR[91,2] = PR[90,2] + -3.916;
   1:L PR[91] R[100]mm/sec CNT100;
   1:  PR[91,1] = PR[90,1] + -7.029;
   1:  PR[91,2] = PR[90,2] + -0.727;
   1:L PR[91] R[100]mm/sec CNT100;
   1:  PR[91,1] = PR[90,1] + -7.293;
   1:  PR[91,2] = PR[90,2] + 2.318;
   1:L PR[91] R[100]mm/sec CNT100;
   1:  PR[91,1] = PR[90,1] + -7.306;
   1:  PR[91,2] = PR[90,2] + 2.433;
   1:L PR[91] R[100]mm/sec CNT100;
   1:  PR[91,1] = PR[90,1] + -8.091;
   1:  PR[91,2] = PR[90,2] + 5.368;
   1:L PR[91] R[100]mm/sec CNT100;
   1:  PR[91,1] = PR[90,1] + -8.129;
   1:  PR[91,2] = PR[90,2] + 5.475;
   1:L PR[91] R[100]mm/sec CNT100;
   1:  PR[91,1] = PR[90,1] + -9.414;
   1:  PR[91,2] = PR[90,2] + 8.233;
   1:L PR[91] R[100]mm/sec CNT100;
   1:  PR[91,1] = PR[90,1] + -9.471;
   1:  PR[91,2] = PR[90,2] + 8.324;
   1:L PR[91] R[100]mm/sec CNT100;
   1:  PR[91,1] = PR[90,1] + -11.219;
   1:  PR[91,2] = PR[90,2] + 10.821;
   1:L PR[91] R[100]mm/sec CNT100;
   1:  PR[91,1] = PR[90,1] + -13.483;
   1:  PR[91,2] = PR[90,2] + 13.085;
   1:L PR[91] R[100]mm/sec CNT100;
   1:  PR[91,1] = PR[90,1] + -15.981;
   1:  PR[91,2] = PR[90,2] + 14.834;
   1:L PR[91] R[100]mm/sec CNT100;
   1:  PR[91,1] = PR[90,1] + -16.060;
   1:  PR[91,2] = PR[90,2] + 14.884;
   1:L PR[91] R[100]mm/sec CNT100;
   1:  PR[91,1] = PR[90,1] + -18.835;
   1:  PR[91,2] = PR[90,2] + 16.178;
   1:L PR[91] R[100]mm/sec CNT100;
   1:  PR[91,1] = PR[90,1] + -18.912;
   1:  PR[91,2] = PR[90,2] + 16.205;
   1:L PR[91] R[100]mm/sec CNT100;
   1:  PR[91,1] = PR[90,1] + -21.856;
   1:  PR[91,2] = PR[90,2] + 16.994;
   1:L PR[91] R[100]mm/sec CNT100;
   1:  PR[91,1] = PR[90,1] + -25.040;
   1:  PR[91,2] = PR[90,2] + 17.278;
   1:L PR[91] R[100]mm/sec CNT100;
   1:  PR[91,1] = PR[90,1] + -28.125;
   1:  PR[91,2] = PR[90,2] + 17.008;
   1:L PR[91] R[100]mm/sec CNT100;
   1:  PR[91,1] = PR[90,1] + -28.191;
   1:  PR[91,2] = PR[90,2] + 17.001;
   1:L PR[91] R[100]mm/sec CNT100;
   1:  PR[91,1] = PR[90,1] + -31.169;
   1:  PR[91,2] = PR[90,2] + 16.202;
   1:L PR[91] R[100]mm/sec CNT100;
   1:  PR[91,1] = PR[90,1] + -31.222;
   1:  PR[91,2] = PR[90,2] + 16.184;
   1:L PR[91] R[100]mm/sec CNT100;
   1:  PR[91,1] = PR[90,1] + -33.981;
   1:  PR[91,2] = PR[90,2] + 14.897;
   1:L PR[91] R[100]mm/sec CNT100;
   1:  PR[91,1] = PR[90,1] + -36.597;
   1:  PR[91,2] = PR[90,2] + 13.076;
   1:L PR[91] R[100]mm/sec CNT100;
   1:  PR[91,1] = PR[90,1] + -38.849;
   1:  PR[91,2] = PR[90,2] + 10.823;
   1:L PR[91] R[100]mm/sec CNT100TB   .50sec,CALL END_PUD;
   1:  PR[92] = PR[91];
   1:  PR[92,3] = PR[92,3] + 20;
   1:J PR[92] 10% FINE;
   1:  PR[91,1] = PR[90,1] + -92.766;
   1:  PR[91,2] = PR[90,2] + -3.793;
   1:  PR[92] = PR[91];
   1:  PR[92,3] = PR[92,3] + 20;
   1:J PR[92] 10% FINE;
   1:L PR[91] R[100]mm/sec CNT100;
   1:  CALL LASER_DRAHT_START;
   1:  PR[91,1] = PR[90,1] + -92.759;
   1:  PR[91,2] = PR[90,2] + -3.859;
   1:L PR[91] R[100]mm/sec CNT100;
   1:  PR[91,1] = PR[90,1] + -91.954;
   1:  PR[91,2] = PR[90,2] + -6.864;
   1:L PR[91] R[100]mm/sec CNT100;
   1:  PR[91,1] = PR[90,1] + -91.939;
   1:  PR[91,2] = PR[90,2] + -6.910;
   1:L PR[91] R[100]mm/sec CNT100;
   1:  PR[91,1] = PR[90,1] + -90.633;
   1:  PR[91,2] = PR[90,2] + -9.710;
   1:L PR[91] R[100]mm/sec CNT100;
   1:  PR[91,1] = PR[90,1] + -90.607;
   1:  PR[91,2] = PR[90,2] + -9.756;
   1:L PR[91] R[100]mm/sec CNT100;
   1:  PR[91,1] = PR[90,1] + -88.831;
   1:  PR[91,2] = PR[90,2] + -12.290;
   1:L PR[91] R[100]mm/sec CNT100;
   1:  PR[91,1] = PR[90,1] + -88.791;
   1:  PR[91,2] = PR[90,2] + -12.335;
   1:L PR[91] R[100]mm/sec CNT100;
   1:  PR[91,1] = PR[90,1] + -86.615;
   1:  PR[91,2] = PR[90,2] + -14.509;
   1:L PR[91] R[100]mm/sec CNT100;
   1:  PR[91,1] = PR[90,1] + -86.558;
   1:  PR[91,2] = PR[90,2] + -14.551;
   1:L PR[91] R[100]mm/sec CNT100;
   1:  PR[91,1] = PR[90,1] + -84.025;
   1:  PR[91,2] = PR[90,2] + -16.323;
   1:L PR[91] R[100]mm/sec CNT100;
   1:  PR[91,1] = PR[90,1] + -81.224;
   1:  PR[91,2] = PR[90,2] + -17.628;
   1:L PR[91] R[100]mm/sec CNT100;
   1:  PR[91,1] = PR[90,1] + -81.158;
   1:  PR[91,2] = PR[90,2] + -17.658;
   1:L PR[91] R[100]mm/sec CNT100;
   1:  PR[91,1] = PR[90,1] + -78.196;
   1:  PR[91,2] = PR[90,2] + -18.450;
   1:L PR[91] R[100]mm/sec CNT100;
   1:  PR[91,1] = PR[90,1] + -78.111;
   1:  PR[91,2] = PR[90,2] + -18.469;
   1:L PR[91] R[100]mm/sec CNT100;
   1:  PR[91,1] = PR[90,1] + -75.070;
   1:  PR[91,2] = PR[90,2] + -18.733;
   1:L PR[91] R[100]mm/sec CNT100;
   1:  PR[91,1] = PR[90,1] + -74.967;
   1:  PR[91,2] = PR[90,2] + -18.734;
   1:L PR[91] R[100]mm/sec CNT100;
   1:  PR[91,1] = PR[90,1] + -71.939;
   1:  PR[91,2] = PR[90,2] + -18.468;
   1:L PR[91] R[100]mm/sec CNT100;
   1:  PR[91,1] = PR[90,1] + -71.821;
   1:  PR[91,2] = PR[90,2] + -18.443;
   1:L PR[91] R[100]mm/sec CNT100;
   1:  PR[91,1] = PR[90,1] + -68.914;
   1:  PR[91,2] = PR[90,2] + -17.663;
   1:L PR[91] R[100]mm/sec CNT100;
   1:  PR[91,1] = PR[90,1] + -66.028;
   1:  PR[91,2] = PR[90,2] + -16.323;
   1:L PR[91] R[100]mm/sec CNT100;
   1:  PR[91,1] = PR[90,1] + -63.413;
   1:  PR[91,2] = PR[90,2] + -14.487;
   1:L PR[91] R[100]mm/sec CNT100;
   1:  PR[91,1] = PR[90,1] + -61.305;
   1:  PR[91,2] = PR[90,2] + -12.379;
   1:L PR[91] R[100]mm/sec CNT100;
   1:  PR[91,1] = PR[90,1] + -61.195;
   1:  PR[91,2] = PR[90,2] + -12.257;
   1:L PR[91] R[100]mm/sec CNT100;
   1:  PR[91,1] = PR[90,1] + -59.478;
   1:  PR[91,2] = PR[90,2] + -9.805;
   1:L PR[91] R[100]mm/sec CNT100;
   1:  PR[91,1] = PR[90,1] + -59.387;
   1:  PR[91,2] = PR[90,2] + -9.648;
   1:L PR[91] R[100]mm/sec CNT100;
   1:  PR[91,1] = PR[90,1] + -58.130;
   1:  PR[91,2] = PR[90,2] + -6.952;
   1:L PR[91] R[100]mm/sec CNT100;
   1:  PR[91,1] = PR[90,1] + -58.071;
   1:  PR[91,2] = PR[90,2] + -6.770;
   1:L PR[91] R[100]mm/sec CNT100;
   1:  PR[91,1] = PR[90,1] + -57.306;
   1:  PR[91,2] = PR[90,2] + -3.913;
   1:L PR[91] R[100]mm/sec CNT100;
   1:  PR[91,1] = PR[90,1] + -57.026;
   1:  PR[91,2] = PR[90,2] + -0.729;
   1:L PR[91] R[100]mm/sec CNT100;
   1:  PR[91,1] = PR[90,1] + -57.283;
   1:  PR[91,2] = PR[90,2] + 2.208;
   1:L PR[91] R[100]mm/sec CNT100;
   1:  PR[91,1] = PR[90,1] + -57.308;
   1:  PR[91,2] = PR[90,2] + 2.443;
   1:L PR[91] R[100]mm/sec CNT100;
   1:  PR[91,1] = PR[90,1] + -58.070;
   1:  PR[91,2] = PR[90,2] + 5.287;
   1:L PR[91] R[100]mm/sec CNT100;
   1:  PR[91,1] = PR[90,1] + -58.141;
   1:  PR[91,2] = PR[90,2] + 5.507;
   1:L PR[91] R[100]mm/sec CNT100;
   1:  PR[91,1] = PR[90,1] + -59.385;
   1:  PR[91,2] = PR[90,2] + 8.175;
   1:L PR[91] R[100]mm/sec CNT100;
   1:  PR[91,1] = PR[90,1] + -59.495;
   1:  PR[91,2] = PR[90,2] + 8.364;
   1:L PR[91] R[100]mm/sec CNT100;
   1:  PR[91,1] = PR[90,1] + -61.196;
   1:  PR[91,2] = PR[90,2] + 10.791;
   1:L PR[91] R[100]mm/sec CNT100;
   1:  PR[91,1] = PR[90,1] + -61.331;
   1:  PR[91,2] = PR[90,2] + 10.941;
   1:L PR[91] R[100]mm/sec CNT100;
   1:  PR[91,1] = PR[90,1] + -63.418;
   1:  PR[91,2] = PR[90,2] + 13.027;
   1:L PR[91] R[100]mm/sec CNT100;
   1:  PR[91,1] = PR[90,1] + -66.039;
   1:  PR[91,2] = PR[90,2] + 14.867;
   1:L PR[91] R[100]mm/sec CNT100;
   1:  PR[91,1] = PR[90,1] + -68.932;
   1:  PR[91,2] = PR[90,2] + 16.208;
   1:L PR[91] R[100]mm/sec CNT100;
   1:  PR[91,1] = PR[90,1] + -71.816;
   1:  PR[91,2] = PR[90,2] + 16.980;
   1:L PR[91] R[100]mm/sec CNT100;
   1:  PR[91,1] = PR[90,1] + -71.967;
   1:  PR[91,2] = PR[90,2] + 17.011;
   1:L PR[91] R[100]mm/sec CNT100;
   1:  PR[91,1] = PR[90,1] + -74.969;
   1:  PR[91,2] = PR[90,2] + 17.273;
   1:L PR[91] R[100]mm/sec CNT100;
   1:  PR[91,1] = PR[90,1] + -75.103;
   1:L PR[91] R[100]mm/sec CNT100;
   1:  PR[91,1] = PR[90,1] + -78.117;
   1:  PR[91,2] = PR[90,2] + 17.008;
   1:L PR[91] R[100]mm/sec CNT100;
   1:  PR[91,1] = PR[90,1] + -78.231;
   1:  PR[91,2] = PR[90,2] + 16.984;
   1:L PR[91] R[100]mm/sec CNT100;
   1:  PR[91,1] = PR[90,1] + -81.153;
   1:  PR[91,2] = PR[90,2] + 16.200;
   1:L PR[91] R[100]mm/sec CNT100;
   1:  PR[91,1] = PR[90,1] + -84.035;
   1:  PR[91,2] = PR[90,2] + 14.860;
   1:L PR[91] R[100]mm/sec CNT100;
   1:  PR[91,1] = PR[90,1] + -86.640;
   1:  PR[91,2] = PR[90,2] + 13.030;
   1:L PR[91] R[100]mm/sec CNT100;
   1:  PR[91,1] = PR[90,1] + -88.786;
   1:  PR[91,2] = PR[90,2] + 10.884;
   1:L PR[91] R[100]mm/sec CNT100;
   1:  PR[91,1] = PR[90,1] + -88.844;
   1:  PR[91,2] = PR[90,2] + 10.820;
   1:L PR[91] R[100]mm/sec CNT100;
   1:  PR[91,1] = PR[90,1] + -90.605;
   1:  PR[91,2] = PR[90,2] + 8.304;
   1:L PR[91] R[100]mm/sec CNT100;
   1:  PR[91,1] = PR[90,1] + -90.644;
   1:  PR[91,2] = PR[90,2] + 8.236;
   1:L PR[91] R[100]mm/sec CNT100;
   1:  PR[91,1] = PR[90,1] + -91.940;
   1:  PR[91,2] = PR[90,2] + 5.457;
   1:L PR[91] R[100]mm/sec CNT100;
   1:  PR[91,1] = PR[90,1] + -91.962;
   1:  PR[91,2] = PR[90,2] + 5.387;
   1:L PR[91] R[100]mm/sec CNT100;
   1:  PR[91,1] = PR[90,1] + -92.754;
   1:  PR[91,2] = PR[90,2] + 2.431;
   1:L PR[91] R[100]mm/sec CNT100;
   1:  PR[91,1] = PR[90,1] + -93.034;
   1:  PR[91,2] = PR[90,2] + -0.731;
   1:L PR[91] R[100]mm/sec CNT100;
   1:  PR[91,1] = PR[90,1] + -92.766;
   1:  PR[91,2] = PR[90,2] + -3.793;
   1:L PR[91] R[100]mm/sec CNT100TB   .50sec,CALL END_PUD;
   1:  PR[92] = PR[91];
   1:  PR[92,3] = PR[92,3] + 20;
   1:J PR[92] 10% FINE;
   1:  PR[91] = PR[90];
   1:  PR[91,1] = PR[90,1] + 38.612;
   1:  PR[91,2] = PR[90,2] + 11.034;
   1:  PR[91,3] = PR[90,3] + 10.595;
   1:  PR[92] = PR[91];
   1:  PR[92,3] = PR[92,3] + 20;
   1:J PR[92] 10% FINE;
   1:L PR[91] R[100]mm/sec CNT100;
   1:  CALL LASER_DRAHT_START;
   1:  PR[91,1] = PR[90,1] + 36.655;
   1:  PR[91,2] = PR[90,2] + 12.990;
   1:L PR[91] R[100]mm/sec CNT100;
   1:  PR[91,1] = PR[90,1] + 36.236;
   1:  PR[91,2] = PR[90,2] + 13.313;
   1:L PR[91] R[100]mm/sec CNT100;
   1:  PR[91,1] = PR[90,1] + 33.931;
   1:  PR[91,2] = PR[90,2] + 14.925;
   1:L PR[91] R[100]mm/sec CNT100;
   1:  PR[91,1] = PR[90,1] + 31.385;
   1:  PR[91,2] = PR[90,2] + 16.111;
   1:L PR[91] R[100]mm/sec CNT100;
   1:  PR[91,1] = PR[90,1] + 30.892;
   1:  PR[91,2] = PR[90,2] + 16.316;
   1:L PR[91] R[100]mm/sec CNT100;
   1:  PR[91,1] = PR[90,1] + 28.221;
   1:  PR[91,2] = PR[90,2] + 17.031;
   1:L PR[91] R[100]mm/sec CNT100;
   1:  PR[91,1] = PR[90,1] + 27.682;
   1:  PR[91,2] = PR[90,2] + 17.103;
   1:L PR[91] R[100]mm/sec CNT100;
   1:  PR[91,1] = PR[90,1] + 24.895;
   1:  PR[91,2] = PR[90,2] + 17.346;
   1:L PR[91] R[100]mm/sec CNT100;
   1:  PR[91,1] = PR[90,1] + 22.105;
   1:  PR[91,2] = PR[90,2] + 17.101;
   1:L PR[91] R[100]mm/sec CNT100;
   1:  PR[91,1] = PR[90,1] + 21.561;
   1:  PR[91,2] = PR[90,2] + 17.030;
   1:L PR[91] R[100]mm/sec CNT100;
   1:  PR[91,1] = PR[90,1] + 18.946;
   1:  PR[91,2] = PR[90,2] + 16.329;
   1:L PR[91] R[100]mm/sec CNT100;
   1:  PR[91,1] = PR[90,1] + 16.336;
   1:  PR[91,2] = PR[90,2] + 15.111;
   1:L PR[91] R[100]mm/sec CNT100;
   1:  PR[91,1] = PR[90,1] + 15.825;
   1:  PR[91,2] = PR[90,2] + 14.900;
   1:L PR[91] R[100]mm/sec CNT100;
   1:  PR[91,1] = PR[90,1] + 13.572;
   1:  PR[91,2] = PR[90,2] + 13.323;
   1:L PR[91] R[100]mm/sec CNT100;
   1:  PR[91,1] = PR[90,1] + 13.124;
   1:  PR[91,2] = PR[90,2] + 12.981;
   1:L PR[91] R[100]mm/sec CNT100;
   1:  PR[91,1] = PR[90,1] + 11.189;
   1:  PR[91,2] = PR[90,2] + 11.045;
   1:L PR[91] R[100]mm/sec CNT100;
   1:  PR[91,1] = PR[90,1] + 10.840;
   1:  PR[91,2] = PR[90,2] + 10.592;
   1:L PR[91] R[100]mm/sec CNT100;
   1:  PR[91,1] = PR[90,1] + 9.242;
   1:  PR[91,2] = PR[90,2] + 8.308;
   1:L PR[91] R[100]mm/sec CNT100;
   1:  PR[91,1] = PR[90,1] + 8.066;
   1:  PR[91,2] = PR[90,2] + 5.787;
   1:L PR[91] R[100]mm/sec CNT100;
   1:  PR[91,1] = PR[90,1] + 7.846;
   1:  PR[91,2] = PR[90,2] + 5.257;
   1:L PR[91] R[100]mm/sec CNT100;
   1:  PR[91,1] = PR[90,1] + 7.148;
   1:  PR[91,2] = PR[90,2] + 2.652;
   1:L PR[91] R[100]mm/sec CNT100;
   1:  PR[91,1] = PR[90,1] + 6.899;
   1:  PR[91,2] = PR[90,2] + -0.200;
   1:L PR[91] R[100]mm/sec CNT100;
   1:  PR[91,1] = PR[90,1] + 6.825;
   1:  PR[91,2] = PR[90,2] + -0.772;
   1:L PR[91] R[100]mm/sec CNT100;
   1:  PR[91,1] = PR[90,1] + 7.065;
   1:  PR[91,2] = PR[90,2] + -3.525;
   1:L PR[91] R[100]mm/sec CNT100;
   1:  PR[91,1] = PR[90,1] + 7.137;
   1:  PR[91,2] = PR[90,2] + -4.068;
   1:L PR[91] R[100]mm/sec CNT100;
   1:  PR[91,1] = PR[90,1] + 7.847;
   1:  PR[91,2] = PR[90,2] + -6.717;
   1:L PR[91] R[100]mm/sec CNT100;
   1:  PR[91,1] = PR[90,1] + 8.067;
   1:  PR[91,2] = PR[90,2] + -7.248;
   1:L PR[91] R[100]mm/sec CNT100;
   1:  PR[91,1] = PR[90,1] + 9.243;
   1:  PR[91,2] = PR[90,2] + -9.770;
   1:L PR[91] R[100]mm/sec CNT100;
   1:  PR[91,1] = PR[90,1] + 10.843;
   1:  PR[91,2] = PR[90,2] + -12.054;
   1:L PR[91] R[100]mm/sec CNT100;
   1:  PR[91,1] = PR[90,1] + 11.192;
   1:  PR[91,2] = PR[90,2] + -12.507;
   1:L PR[91] R[100]mm/sec CNT100;
   1:  PR[91,1] = PR[90,1] + 13.129;
   1:  PR[91,2] = PR[90,2] + -14.443;
   1:L PR[91] R[100]mm/sec CNT100;
   1:  PR[91,1] = PR[90,1] + 13.577;
   1:  PR[91,2] = PR[90,2] + -14.786;
   1:L PR[91] R[100]mm/sec CNT100;
   1:  PR[91,1] = PR[90,1] + 15.868;
   1:  PR[91,2] = PR[90,2] + -16.389;
   1:L PR[91] R[100]mm/sec CNT100;
   1:  PR[91,1] = PR[90,1] + 18.394;
   1:  PR[91,2] = PR[90,2] + -17.566;
   1:L PR[91] R[100]mm/sec CNT100;
   1:  PR[91,1] = PR[90,1] + 18.911;
   1:  PR[91,2] = PR[90,2] + -17.779;
   1:L PR[91] R[100]mm/sec CNT100;
   1:  PR[91,1] = PR[90,1] + 21.572;
   1:  PR[91,2] = PR[90,2] + -18.491;
   1:L PR[91] R[100]mm/sec CNT100;
   1:  PR[91,1] = PR[90,1] + 22.116;
   1:  PR[91,2] = PR[90,2] + -18.562;
   1:L PR[91] R[100]mm/sec CNT100;
   1:  PR[91,1] = PR[90,1] + 24.906;
   1:  PR[91,2] = PR[90,2] + -18.805;
   1:L PR[91] R[100]mm/sec CNT100;
   1:  PR[91,1] = PR[90,1] + 27.693;
   1:  PR[91,2] = PR[90,2] + -18.560;
   1:L PR[91] R[100]mm/sec CNT100;
   1:  PR[91,1] = PR[90,1] + 28.232;
   1:  PR[91,2] = PR[90,2] + -18.488;
   1:L PR[91] R[100]mm/sec CNT100;
   1:  PR[91,1] = PR[90,1] + 30.860;
   1:  PR[91,2] = PR[90,2] + -17.783;
   1:L PR[91] R[100]mm/sec CNT100;
   1:  PR[91,1] = PR[90,1] + 33.475;
   1:  PR[91,2] = PR[90,2] + -16.563;
   1:L PR[91] R[100]mm/sec CNT100;
   1:  PR[91,1] = PR[90,1] + 33.971;
   1:  PR[91,2] = PR[90,2] + -16.357;
   1:L PR[91] R[100]mm/sec CNT100;
   1:  PR[91,1] = PR[90,1] + 36.240;
   1:  PR[91,2] = PR[90,2] + -14.768;
   1:L PR[91] R[100]mm/sec CNT100;
   1:  PR[91,1] = PR[90,1] + 36.659;
   1:  PR[91,2] = PR[90,2] + -14.445;
   1:L PR[91] R[100]mm/sec CNT100;
   1:  PR[91,1] = PR[90,1] + 38.615;
   1:  PR[91,2] = PR[90,2] + -12.490;
   1:L PR[91] R[100]mm/sec CNT100;
   1:  PR[91,1] = PR[90,1] + 38.932;
   1:  PR[91,2] = PR[90,2] + -12.075;
   1:L PR[91] R[100]mm/sec CNT100;
   1:  PR[91,1] = PR[90,1] + 40.552;
   1:  PR[91,2] = PR[90,2] + -9.762;
   1:L PR[91] R[100]mm/sec CNT100;
   1:  PR[91,1] = PR[90,1] + 41.741;
   1:  PR[91,2] = PR[90,2] + -7.212;
   1:L PR[91] R[100]mm/sec CNT100;
   1:  PR[91,1] = PR[90,1] + 41.939;
   1:  PR[91,2] = PR[90,2] + -6.732;
   1:L PR[91] R[100]mm/sec CNT100;
   1:  PR[91,1] = PR[90,1] + 42.647;
   1:  PR[91,2] = PR[90,2] + -4.089;
   1:L PR[91] R[100]mm/sec CNT100;
   1:  PR[91,1] = PR[90,1] + 42.898;
   1:  PR[91,2] = PR[90,2] + -1.213;
   1:L PR[91] R[100]mm/sec CNT100;
   1:  PR[91,1] = PR[90,1] + 42.958;
   1:  PR[91,2] = PR[90,2] + -0.697;
   1:L PR[91] R[100]mm/sec CNT100;
   1:  PR[91,1] = PR[90,1] + 42.725;
   1:  PR[91,2] = PR[90,2] + 2.078;
   1:L PR[91] R[100]mm/sec CNT100;
   1:  PR[91,1] = PR[90,1] + 42.658;
   1:  PR[91,2] = PR[90,2] + 2.588;
   1:L PR[91] R[100]mm/sec CNT100;
   1:  PR[91,1] = PR[90,1] + 41.938;
   1:  PR[91,2] = PR[90,2] + 5.275;
   1:L PR[91] R[100]mm/sec CNT100;
   1:  PR[91,1] = PR[90,1] + 41.740;
   1:  PR[91,2] = PR[90,2] + 5.755;
   1:L PR[91] R[100]mm/sec CNT100;
   1:  PR[91,1] = PR[90,1] + 40.550;
   1:  PR[91,2] = PR[90,2] + 8.306;
   1:L PR[91] R[100]mm/sec CNT100;
   1:  PR[91,1] = PR[90,1] + 38.929;
   1:  PR[91,2] = PR[90,2] + 10.620;
   1:L PR[91] R[100]mm/sec CNT100;
   1:  PR[91,1] = PR[90,1] + 38.612;
   1:  PR[91,2] = PR[90,2] + 11.034;
   1:L PR[91] R[100]mm/sec CNT100TB   .50sec,CALL END_PUD;
   1:  PR[92] = PR[91];
   1:  PR[92,3] = PR[92,3] + 20;
   1:J PR[92] 10% FINE;
   1:  PR[91,1] = PR[90,1] + 68.240;
   1:  PR[91,2] = PR[90,2] + 16.079;
   1:  PR[92] = PR[91];
   1:  PR[92,3] = PR[92,3] + 20;
   1:J PR[92] 10% FINE;
   1:L PR[91] R[100]mm/sec CNT100;
   1:  CALL LASER_DRAHT_START;
   1:  PR[91,1] = PR[90,1] + 66.074;
   1:  PR[91,2] = PR[90,2] + 15.070;
   1:L PR[91] R[100]mm/sec CNT100;
   1:  PR[91,1] = PR[90,1] + 65.222;
   1:  PR[91,2] = PR[90,2] + 14.539;
   1:L PR[91] R[100]mm/sec CNT100;
   1:  PR[91,1] = PR[90,1] + 63.304;
   1:  PR[91,2] = PR[90,2] + 13.197;
   1:L PR[91] R[100]mm/sec CNT100;
   1:  PR[91,1] = PR[90,1] + 60.881;
   1:  PR[91,2] = PR[90,2] + 10.783;
   1:L PR[91] R[100]mm/sec CNT100;
   1:  PR[91,1] = PR[90,1] + 59.564;
   1:  PR[91,2] = PR[90,2] + 8.902;
   1:L PR[91] R[100]mm/sec CNT100;
   1:  PR[91,1] = PR[90,1] + 58.970;
   1:  PR[91,2] = PR[90,2] + 7.963;
   1:L PR[91] R[100]mm/sec CNT100;
   1:  PR[91,1] = PR[90,1] + 58.021;
   1:  PR[91,2] = PR[90,2] + 5.928;
   1:L PR[91] R[100]mm/sec CNT100;
   1:  PR[91,1] = PR[90,1] + 57.634;
   1:  PR[91,2] = PR[90,2] + 4.827;
   1:L PR[91] R[100]mm/sec CNT100;
   1:  PR[91,1] = PR[90,1] + 57.065;
   1:  PR[91,2] = PR[90,2] + 2.704;
   1:L PR[91] R[100]mm/sec CNT100;
   1:  PR[91,1] = PR[90,1] + 56.866;
   1:  PR[91,2] = PR[90,2] + 0.422;
   1:L PR[91] R[100]mm/sec CNT100;
   1:  PR[91,1] = PR[90,1] + 56.733;
   1:  PR[91,2] = PR[90,2] + -0.755;
   1:L PR[91] R[100]mm/sec CNT100;
   1:  PR[91,1] = PR[90,1] + 56.924;
   1:  PR[91,2] = PR[90,2] + -2.946;
   1:L PR[91] R[100]mm/sec CNT100;
   1:  PR[91,1] = PR[90,1] + 57.059;
   1:  PR[91,2] = PR[90,2] + -4.139;
   1:L PR[91] R[100]mm/sec CNT100;
   1:  PR[91,1] = PR[90,1] + 57.633;
   1:  PR[91,2] = PR[90,2] + -6.284;
   1:L PR[91] R[100]mm/sec CNT100;
   1:  PR[91,1] = PR[90,1] + 58.021;
   1:  PR[91,2] = PR[90,2] + -7.386;
   1:L PR[91] R[100]mm/sec CNT100;
   1:  PR[91,1] = PR[90,1] + 58.969;
   1:  PR[91,2] = PR[90,2] + -9.420;
   1:L PR[91] R[100]mm/sec CNT100;
   1:  PR[91,1] = PR[90,1] + 59.563;
   1:  PR[91,2] = PR[90,2] + -10.359;
   1:L PR[91] R[100]mm/sec CNT100;
   1:  PR[91,1] = PR[90,1] + 60.880;
   1:  PR[91,2] = PR[90,2] + -12.240;
   1:L PR[91] R[100]mm/sec CNT100;
   1:  PR[91,1] = PR[90,1] + 62.527;
   1:  PR[91,2] = PR[90,2] + -13.887;
   1:L PR[91] R[100]mm/sec CNT100;
   1:  PR[91,1] = PR[90,1] + 63.298;
   1:  PR[91,2] = PR[90,2] + -14.651;
   1:L PR[91] R[100]mm/sec CNT100;
   1:  PR[91,1] = PR[90,1] + 65.216;
   1:  PR[91,2] = PR[90,2] + -15.995;
   1:L PR[91] R[100]mm/sec CNT100;
   1:  PR[91,1] = PR[90,1] + 66.068;
   1:  PR[91,2] = PR[90,2] + -16.526;
   1:L PR[91] R[100]mm/sec CNT100;
   1:  PR[91,1] = PR[90,1] + 68.232;
   1:  PR[91,2] = PR[90,2] + -17.535;
   1:L PR[91] R[100]mm/sec CNT100;
   1:  PR[91,1] = PR[90,1] + 69.100;
   1:  PR[91,2] = PR[90,2] + -17.835;
   1:L PR[91] R[100]mm/sec CNT100;
   1:  PR[91,1] = PR[90,1] + 71.443;
   1:  PR[91,2] = PR[90,2] + -18.463;
   1:L PR[91] R[100]mm/sec CNT100;
   1:  PR[91,1] = PR[90,1] + 73.947;
   1:  PR[91,2] = PR[90,2] + -18.683;
   1:L PR[91] R[100]mm/sec CNT100;
   1:  PR[91,1] = PR[90,1] + 74.828;
   1:  PR[91,2] = PR[90,2] + -18.778;
   1:L PR[91] R[100]mm/sec CNT100;
   1:  PR[91,1] = PR[90,1] + 77.314;
   1:  PR[91,2] = PR[90,2] + -18.561;
   1:L PR[91] R[100]mm/sec CNT100;
   1:  PR[91,1] = PR[90,1] + 78.117;
   1:  PR[91,2] = PR[90,2] + -18.467;
   1:L PR[91] R[100]mm/sec CNT100;
   1:  PR[91,1] = PR[90,1] + 80.574;
   1:  PR[91,2] = PR[90,2] + -17.810;
   1:L PR[91] R[100]mm/sec CNT100;
   1:  PR[91,1] = PR[90,1] + 81.275;
   1:  PR[91,2] = PR[90,2] + -17.562;
   1:L PR[91] R[100]mm/sec CNT100;
   1:  PR[91,1] = PR[90,1] + 83.607;
   1:  PR[91,2] = PR[90,2] + -16.475;
   1:L PR[91] R[100]mm/sec CNT100;
   1:  PR[91,1] = PR[90,1] + 84.190;
   1:  PR[91,2] = PR[90,2] + -16.106;
   1:L PR[91] R[100]mm/sec CNT100;
   1:  PR[91,1] = PR[90,1] + 86.332;
   1:  PR[91,2] = PR[90,2] + -14.608;
   1:L PR[91] R[100]mm/sec CNT100;
   1:  PR[91,1] = PR[90,1] + 88.207;
   1:  PR[91,2] = PR[90,2] + -12.734;
   1:L PR[91] R[100]mm/sec CNT100;
   1:  PR[91,1] = PR[90,1] + 88.680;
   1:  PR[91,2] = PR[90,2] + -12.258;
   1:L PR[91] R[100]mm/sec CNT100;
   1:  PR[91,1] = PR[90,1] + 90.193;
   1:  PR[91,2] = PR[90,2] + -10.098;
   1:L PR[91] R[100]mm/sec CNT100;
   1:  PR[91,1] = PR[90,1] + 90.532;
   1:  PR[91,2] = PR[90,2] + -9.557;
   1:L PR[91] R[100]mm/sec CNT100;
   1:  PR[91,1] = PR[90,1] + 91.651;
   1:  PR[91,2] = PR[90,2] + -7.159;
   1:L PR[91] R[100]mm/sec CNT100;
   1:  PR[91,1] = PR[90,1] + 91.854;
   1:  PR[91,2] = PR[90,2] + -6.576;
   1:L PR[91] R[100]mm/sec CNT100;
   1:  PR[91,1] = PR[90,1] + 92.536;
   1:  PR[91,2] = PR[90,2] + -4.029;
   1:L PR[91] R[100]mm/sec CNT100;
   1:  PR[91,1] = PR[90,1] + 92.773;
   1:  PR[91,2] = PR[90,2] + -1.313;
   1:L PR[91] R[100]mm/sec CNT100;
   1:  PR[91,1] = PR[90,1] + 92.841;
   1:  PR[91,2] = PR[90,2] + -0.706;
   1:L PR[91] R[100]mm/sec CNT100;
   1:  PR[91,1] = PR[90,1] + 92.608;
   1:  PR[91,2] = PR[90,2] + 1.952;
   1:L PR[91] R[100]mm/sec CNT100;
   1:  PR[91,1] = PR[90,1] + 92.542;
   1:  PR[91,2] = PR[90,2] + 2.547;
   1:L PR[91] R[100]mm/sec CNT100;
   1:  PR[91,1] = PR[90,1] + 91.854;
   1:  PR[91,2] = PR[90,2] + 5.116;
   1:L PR[91] R[100]mm/sec CNT100;
   1:  PR[91,1] = PR[90,1] + 91.651;
   1:  PR[91,2] = PR[90,2] + 5.698;
   1:L PR[91] R[100]mm/sec CNT100;
   1:  PR[91,1] = PR[90,1] + 90.534;
   1:  PR[91,2] = PR[90,2] + 8.095;
   1:L PR[91] R[100]mm/sec CNT100;
   1:  PR[91,1] = PR[90,1] + 90.195;
   1:  PR[91,2] = PR[90,2] + 8.637;
   1:L PR[91] R[100]mm/sec CNT100;
   1:  PR[91,1] = PR[90,1] + 88.684;
   1:  PR[91,2] = PR[90,2] + 10.794;
   1:L PR[91] R[100]mm/sec CNT100;
   1:  PR[91,1] = PR[90,1] + 86.335;
   1:  PR[91,2] = PR[90,2] + 13.146;
   1:L PR[91] R[100]mm/sec CNT100;
   1:  PR[91,1] = PR[90,1] + 84.196;
   1:  PR[91,2] = PR[90,2] + 14.644;
   1:L PR[91] R[100]mm/sec CNT100;
   1:  PR[91,1] = PR[90,1] + 83.613;
   1:  PR[91,2] = PR[90,2] + 15.013;
   1:L PR[91] R[100]mm/sec CNT100;
   1:  PR[91,1] = PR[90,1] + 81.283;
   1:  PR[91,2] = PR[90,2] + 16.100;
   1:L PR[91] R[100]mm/sec CNT100;
   1:  PR[91,1] = PR[90,1] + 80.582;
   1:  PR[91,2] = PR[90,2] + 16.348;
   1:L PR[91] R[100]mm/sec CNT100;
   1:  PR[91,1] = PR[90,1] + 78.156;
   1:  PR[91,2] = PR[90,2] + 16.999;
   1:L PR[91] R[100]mm/sec CNT100;
   1:  PR[91,1] = PR[90,1] + 75.548;
   1:  PR[91,2] = PR[90,2] + 17.228;
   1:L PR[91] R[100]mm/sec CNT100;
   1:  PR[91,1] = PR[90,1] + 74.788;
   1:  PR[91,2] = PR[90,2] + 17.318;
   1:L PR[91] R[100]mm/sec CNT100;
   1:  PR[91,1] = PR[90,1] + 72.305;
   1:  PR[91,2] = PR[90,2] + 17.102;
   1:L PR[91] R[100]mm/sec CNT100;
   1:  PR[91,1] = PR[90,1] + 71.473;
   1:  PR[91,2] = PR[90,2] + 17.011;
   1:L PR[91] R[100]mm/sec CNT100;
   1:  PR[91,1] = PR[90,1] + 69.108;
   1:  PR[91,2] = PR[90,2] + 16.379;
   1:L PR[91] R[100]mm/sec CNT100;
   1:  PR[91,1] = PR[90,1] + 68.240;
   1:  PR[91,2] = PR[90,2] + 16.079;
   1:L PR[91] R[100]mm/sec CNT100TB   .50sec,CALL END_PUD;
   1:  PR[92] = PR[91];
   1:  PR[92,3] = PR[92,3] + 20;
   1:J PR[92] 10% FINE;
   1:  PR[91,1] = PR[90,1] + -34.256;
   1:  PR[91,2] = PR[90,2] + 14.708;
   1:  PR[92] = PR[91];
   1:  PR[92,3] = PR[92,3] + 20;
   1:J PR[92] 10% FINE;
   1:L PR[91] R[100]mm/sec CNT100;
   1:  CALL LASER_DRAHT_START;
   1:  PR[91,1] = PR[90,1] + -36.509;
   1:  PR[91,2] = PR[90,2] + 13.130;
   1:L PR[91] R[100]mm/sec CNT100;
   1:  PR[91,1] = PR[90,1] + -38.835;
   1:  PR[91,2] = PR[90,2] + 10.802;
   1:L PR[91] R[100]mm/sec CNT100;
   1:  PR[91,1] = PR[90,1] + -40.418;
   1:  PR[91,2] = PR[90,2] + 8.540;
   1:L PR[91] R[100]mm/sec CNT100;
   1:  PR[91,1] = PR[90,1] + -40.668;
   1:  PR[91,2] = PR[90,2] + 8.142;
   1:L PR[91] R[100]mm/sec CNT100;
   1:  PR[91,1] = PR[90,1] + -41.839;
   1:  PR[91,2] = PR[90,2] + 5.628;
   1:L PR[91] R[100]mm/sec CNT100;
   1:  PR[91,1] = PR[90,1] + -41.991;
   1:  PR[91,2] = PR[90,2] + 5.195;
   1:L PR[91] R[100]mm/sec CNT100;
   1:  PR[91,1] = PR[90,1] + -42.702;
   1:  PR[91,2] = PR[90,2] + 2.536;
   1:L PR[91] R[100]mm/sec CNT100;
   1:  PR[91,1] = PR[90,1] + -42.950;
   1:  PR[91,2] = PR[90,2] + -0.301;
   1:L PR[91] R[100]mm/sec CNT100;
   1:  PR[91,1] = PR[90,1] + -43.001;
   1:  PR[91,2] = PR[90,2] + -0.754;
   1:L PR[91] R[100]mm/sec CNT100;
   1:  PR[91,1] = PR[90,1] + -42.760;
   1:  PR[91,2] = PR[90,2] + -3.519;
   1:L PR[91] R[100]mm/sec CNT100;
   1:  PR[91,1] = PR[90,1] + -42.709;
   1:  PR[91,2] = PR[90,2] + -3.970;
   1:L PR[91] R[100]mm/sec CNT100;
   1:  PR[91,1] = PR[90,1] + -41.991;
   1:  PR[91,2] = PR[90,2] + -6.652;
   1:L PR[91] R[100]mm/sec CNT100;
   1:  PR[91,1] = PR[90,1] + -41.840;
   1:  PR[91,2] = PR[90,2] + -7.086;
   1:L PR[91] R[100]mm/sec CNT100;
   1:  PR[91,1] = PR[90,1] + -40.668;
   1:  PR[91,2] = PR[90,2] + -9.600;
   1:L PR[91] R[100]mm/sec CNT100;
   1:  PR[91,1] = PR[90,1] + -40.419;
   1:  PR[91,2] = PR[90,2] + -9.998;
   1:L PR[91] R[100]mm/sec CNT100;
   1:  PR[91,1] = PR[90,1] + -38.836;
   1:  PR[91,2] = PR[90,2] + -12.260;
   1:L PR[91] R[100]mm/sec CNT100;
   1:  PR[91,1] = PR[90,1] + -36.510;
   1:  PR[91,2] = PR[90,2] + -14.588;
   1:L PR[91] R[100]mm/sec CNT100;
   1:  PR[91,1] = PR[90,1] + -34.257;
   1:  PR[91,2] = PR[90,2] + -16.166;
   1:L PR[91] R[100]mm/sec CNT100;
   1:  PR[91,1] = PR[90,1] + -33.838;
   1:  PR[91,2] = PR[90,2] + -16.431;
   1:L PR[91] R[100]mm/sec CNT100;
   1:  PR[91,1] = PR[90,1] + -31.357;
   1:  PR[91,2] = PR[90,2] + -17.589;
   1:L PR[91] R[100]mm/sec CNT100;
   1:  PR[91,1] = PR[90,1] + -30.864;
   1:  PR[91,2] = PR[90,2] + -17.762;
   1:L PR[91] R[100]mm/sec CNT100;
   1:  PR[91,1] = PR[90,1] + -28.265;
   1:  PR[91,2] = PR[90,2] + -18.460;
   1:L PR[91] R[100]mm/sec CNT100;
   1:  PR[91,1] = PR[90,1] + -25.476;
   1:  PR[91,2] = PR[90,2] + -18.704;
   1:L PR[91] R[100]mm/sec CNT100;
   1:  PR[91,1] = PR[90,1] + -24.947;
   1:  PR[91,2] = PR[90,2] + -18.766;
   1:L PR[91] R[100]mm/sec CNT100;
   1:  PR[91,1] = PR[90,1] + -22.258;
   1:  PR[91,2] = PR[90,2] + -18.530;
   1:L PR[91] R[100]mm/sec CNT100;
   1:  PR[91,1] = PR[90,1] + -21.697;
   1:  PR[91,2] = PR[90,2] + -18.469;
   1:L PR[91] R[100]mm/sec CNT100;
   1:  PR[91,1] = PR[90,1] + -19.110;
   1:  PR[91,2] = PR[90,2] + -17.775;
   1:L PR[91] R[100]mm/sec CNT100;
   1:  PR[91,1] = PR[90,1] + -18.544;
   1:  PR[91,2] = PR[90,2] + -17.579;
   1:L PR[91] R[100]mm/sec CNT100;
   1:  PR[91,1] = PR[90,1] + -16.136;
   1:  PR[91,2] = PR[90,2] + -16.456;
   1:L PR[91] R[100]mm/sec CNT100;
   1:  PR[91,1] = PR[90,1] + -15.600;
   1:  PR[91,2] = PR[90,2] + -16.121;
   1:L PR[91] R[100]mm/sec CNT100;
   1:  PR[91,1] = PR[90,1] + -13.444;
   1:  PR[91,2] = PR[90,2] + -14.611;
   1:L PR[91] R[100]mm/sec CNT100;
   1:  PR[91,1] = PR[90,1] + -11.087;
   1:  PR[91,2] = PR[90,2] + -12.257;
   1:L PR[91] R[100]mm/sec CNT100;
   1:  PR[91,1] = PR[90,1] + -9.587;
   1:  PR[91,2] = PR[90,2] + -10.113;
   1:L PR[91] R[100]mm/sec CNT100;
   1:  PR[91,1] = PR[90,1] + -9.228;
   1:  PR[91,2] = PR[90,2] + -9.544;
   1:L PR[91] R[100]mm/sec CNT100;
   1:  PR[91,1] = PR[90,1] + -8.128;
   1:  PR[91,2] = PR[90,2] + -7.185;
   1:L PR[91] R[100]mm/sec CNT100;
   1:  PR[91,1] = PR[90,1] + -7.898;
   1:  PR[91,2] = PR[90,2] + -6.531;
   1:L PR[91] R[100]mm/sec CNT100;
   1:  PR[91,1] = PR[90,1] + -7.235;
   1:  PR[91,2] = PR[90,2] + -4.052;
   1:L PR[91] R[100]mm/sec CNT100;
   1:  PR[91,1] = PR[90,1] + -7.004;
   1:  PR[91,2] = PR[90,2] + -1.406;
   1:L PR[91] R[100]mm/sec CNT100;
   1:  PR[91,1] = PR[90,1] + -6.931;
   1:  PR[91,2] = PR[90,2] + -0.710;
   1:L PR[91] R[100]mm/sec CNT100;
   1:  PR[91,1] = PR[90,1] + -7.149;
   1:  PR[91,2] = PR[90,2] + 1.873;
   1:L PR[91] R[100]mm/sec CNT100;
   1:  PR[91,1] = PR[90,1] + -7.228;
   1:  PR[91,2] = PR[90,2] + 2.568;
   1:L PR[91] R[100]mm/sec CNT100;
   1:  PR[91,1] = PR[90,1] + -7.898;
   1:  PR[91,2] = PR[90,2] + 5.071;
   1:L PR[91] R[100]mm/sec CNT100;
   1:  PR[91,1] = PR[90,1] + -8.128;
   1:  PR[91,2] = PR[90,2] + 5.725;
   1:L PR[91] R[100]mm/sec CNT100;
   1:  PR[91,1] = PR[90,1] + -9.227;
   1:  PR[91,2] = PR[90,2] + 8.084;
   1:L PR[91] R[100]mm/sec CNT100;
   1:  PR[91,1] = PR[90,1] + -9.586;
   1:  PR[91,2] = PR[90,2] + 8.653;
   1:L PR[91] R[100]mm/sec CNT100;
   1:  PR[91,1] = PR[90,1] + -11.087;
   1:  PR[91,2] = PR[90,2] + 10.797;
   1:L PR[91] R[100]mm/sec CNT100;
   1:  PR[91,1] = PR[90,1] + -13.443;
   1:  PR[91,2] = PR[90,2] + 13.152;
   1:L PR[91] R[100]mm/sec CNT100;
   1:  PR[91,1] = PR[90,1] + -15.598;
   1:  PR[91,2] = PR[90,2] + 14.661;
   1:L PR[91] R[100]mm/sec CNT100;
   1:  PR[91,1] = PR[90,1] + -16.135;
   1:  PR[91,2] = PR[90,2] + 14.997;
   1:L PR[91] R[100]mm/sec CNT100;
   1:  PR[91,1] = PR[90,1] + -18.543;
   1:  PR[91,2] = PR[90,2] + 16.120;
   1:L PR[91] R[100]mm/sec CNT100;
   1:  PR[91,1] = PR[90,1] + -19.109;
   1:  PR[91,2] = PR[90,2] + 16.316;
   1:L PR[91] R[100]mm/sec CNT100;
   1:  PR[91,1] = PR[90,1] + -21.675;
   1:  PR[91,2] = PR[90,2] + 17.004;
   1:L PR[91] R[100]mm/sec CNT100;
   1:  PR[91,1] = PR[90,1] + -24.415;
   1:  PR[91,2] = PR[90,2] + 17.244;
   1:L PR[91] R[100]mm/sec CNT100;
   1:  PR[91,1] = PR[90,1] + -24.997;
   1:  PR[91,2] = PR[90,2] + 17.307;
   1:L PR[91] R[100]mm/sec CNT100;
   1:  PR[91,1] = PR[90,1] + -27.688;
   1:  PR[91,2] = PR[90,2] + 17.072;
   1:L PR[91] R[100]mm/sec CNT100;
   1:  PR[91,1] = PR[90,1] + -28.236;
   1:  PR[91,2] = PR[90,2] + 17.008;
   1:L PR[91] R[100]mm/sec CNT100;
   1:  PR[91,1] = PR[90,1] + -30.863;
   1:  PR[91,2] = PR[90,2] + 16.304;
   1:L PR[91] R[100]mm/sec CNT100;
   1:  PR[91,1] = PR[90,1] + -31.355;
   1:  PR[91,2] = PR[90,2] + 16.131;
   1:L PR[91] R[100]mm/sec CNT100;
   1:  PR[91,1] = PR[90,1] + -33.837;
   1:  PR[91,2] = PR[90,2] + 14.973;
   1:L PR[91] R[100]mm/sec CNT100;
   1:  PR[91,1] = PR[90,1] + -34.256;
   1:  PR[91,2] = PR[90,2] + 14.708;
   1:L PR[91] R[100]mm/sec CNT100TB   .50sec,CALL END_PUD;
   1:  PR[92] = PR[91];
   1:  PR[92,3] = PR[92,3] + 20;
   1:J PR[92] 10% FINE;
   1:  PR[91,1] = PR[90,1] + -91.817;
   1:  PR[91,2] = PR[90,2] + -7.056;
   1:  PR[92] = PR[91];
   1:  PR[92,3] = PR[92,3] + 20;
   1:J PR[92] 10% FINE;
   1:L PR[91] R[100]mm/sec CNT100;
   1:  CALL LASER_DRAHT_START;
   1:  PR[91,1] = PR[90,1] + -90.671;
   1:  PR[91,2] = PR[90,2] + -9.515;
   1:L PR[91] R[100]mm/sec CNT100;
   1:  PR[91,1] = PR[90,1] + -90.415;
   1:  PR[91,2] = PR[90,2] + -9.959;
   1:L PR[91] R[100]mm/sec CNT100;
   1:  PR[91,1] = PR[90,1] + -88.860;
   1:  PR[91,2] = PR[90,2] + -12.177;
   1:L PR[91] R[100]mm/sec CNT100;
   1:  PR[91,1] = PR[90,1] + -88.504;
   1:  PR[91,2] = PR[90,2] + -12.575;
   1:L PR[91] R[100]mm/sec CNT100;
   1:  PR[91,1] = PR[90,1] + -86.607;
   1:  PR[91,2] = PR[90,2] + -14.470;
   1:L PR[91] R[100]mm/sec CNT100;
   1:  PR[91,1] = PR[90,1] + -86.152;
   1:  PR[91,2] = PR[90,2] + -14.802;
   1:L PR[91] R[100]mm/sec CNT100;
   1:  PR[91,1] = PR[90,1] + -83.955;
   1:  PR[91,2] = PR[90,2] + -16.339;
   1:L PR[91] R[100]mm/sec CNT100;
   1:  PR[91,1] = PR[90,1] + -81.527;
   1:  PR[91,2] = PR[90,2] + -17.470;
   1:L PR[91] R[100]mm/sec CNT100;
   1:  PR[91,1] = PR[90,1] + -81.003;
   1:  PR[91,2] = PR[90,2] + -17.705;
   1:L PR[91] R[100]mm/sec CNT100;
   1:  PR[91,1] = PR[90,1] + -78.457;
   1:  PR[91,2] = PR[90,2] + -18.386;
   1:L PR[91] R[100]mm/sec CNT100;
   1:  PR[91,1] = PR[90,1] + -77.855;
   1:  PR[91,2] = PR[90,2] + -18.516;
   1:L PR[91] R[100]mm/sec CNT100;
   1:  PR[91,1] = PR[90,1] + -75.264;
   1:  PR[91,2] = PR[90,2] + -18.741;
   1:L PR[91] R[100]mm/sec CNT100;
   1:  PR[91,1] = PR[90,1] + -74.600;
   1:  PR[91,2] = PR[90,2] + -18.743;
   1:L PR[91] R[100]mm/sec CNT100;
   1:  PR[91,1] = PR[90,1] + -72.046;
   1:  PR[91,2] = PR[90,2] + -18.518;
   1:L PR[91] R[100]mm/sec CNT100;
   1:  PR[91,1] = PR[90,1] + -71.344;
   1:  PR[91,2] = PR[90,2] + -18.371;
   1:L PR[91] R[100]mm/sec CNT100;
   1:  PR[91,1] = PR[90,1] + -68.923;
   1:  PR[91,2] = PR[90,2] + -17.722;
   1:L PR[91] R[100]mm/sec CNT100;
   1:  PR[91,1] = PR[90,1] + -66.589;
   1:  PR[91,2] = PR[90,2] + -16.632;
   1:L PR[91] R[100]mm/sec CNT100;
   1:  PR[91,1] = PR[90,1] + -65.917;
   1:  PR[91,2] = PR[90,2] + -16.336;
   1:L PR[91] R[100]mm/sec CNT100;
   1:  PR[91,1] = PR[90,1] + -63.881;
   1:  PR[91,2] = PR[90,2] + -14.911;
   1:L PR[91] R[100]mm/sec CNT100;
   1:  PR[91,1] = PR[90,1] + -63.238;
   1:  PR[91,2] = PR[90,2] + -14.446;
   1:L PR[91] R[100]mm/sec CNT100;
   1:  PR[91,1] = PR[90,1] + -61.514;
   1:  PR[91,2] = PR[90,2] + -12.723;
   1:L PR[91] R[100]mm/sec CNT100;
   1:  PR[91,1] = PR[90,1] + -60.945;
   1:  PR[91,2] = PR[90,2] + -12.092;
   1:L PR[91] R[100]mm/sec CNT100;
   1:  PR[91,1] = PR[90,1] + -59.562;
   1:  PR[91,2] = PR[90,2] + -10.117;
   1:L PR[91] R[100]mm/sec CNT100;
   1:  PR[91,1] = PR[90,1] + -59.112;
   1:  PR[91,2] = PR[90,2] + -9.341;
   1:L PR[91] R[100]mm/sec CNT100;
   1:  PR[91,1] = PR[90,1] + -58.109;
   1:  PR[91,2] = PR[90,2] + -7.190;
   1:L PR[91] R[100]mm/sec CNT100;
   1:  PR[91,1] = PR[90,1] + -57.821;
   1:  PR[91,2] = PR[90,2] + -6.305;
   1:L PR[91] R[100]mm/sec CNT100;
   1:  PR[91,1] = PR[90,1] + -57.215;
   1:  PR[91,2] = PR[90,2] + -4.041;
   1:L PR[91] R[100]mm/sec CNT100;
   1:  PR[91,1] = PR[90,1] + -56.922;
   1:  PR[91,2] = PR[90,2] + -0.729;
   1:L PR[91] R[100]mm/sec CNT100;
   1:  PR[91,1] = PR[90,1] + -57.119;
   1:  PR[91,2] = PR[90,2] + 1.524;
   1:L PR[91] R[100]mm/sec CNT100;
   1:  PR[91,1] = PR[90,1] + -57.231;
   1:  PR[91,2] = PR[90,2] + 2.585;
   1:L PR[91] R[100]mm/sec CNT100;
   1:  PR[91,1] = PR[90,1] + -57.816;
   1:  PR[91,2] = PR[90,2] + 4.768;
   1:L PR[91] R[100]mm/sec CNT100;
   1:  PR[91,1] = PR[90,1] + -58.141;
   1:  PR[91,2] = PR[90,2] + 5.767;
   1:L PR[91] R[100]mm/sec CNT100;
   1:  PR[91,1] = PR[90,1] + -59.103;
   1:  PR[91,2] = PR[90,2] + 7.830;
   1:L PR[91] R[100]mm/sec CNT100;
   1:  PR[91,1] = PR[90,1] + -59.611;
   1:  PR[91,2] = PR[90,2] + 8.707;
   1:L PR[91] R[100]mm/sec CNT100;
   1:  PR[91,1] = PR[90,1] + -60.940;
   1:  PR[91,2] = PR[90,2] + 10.604;
   1:L PR[91] R[100]mm/sec CNT100;
   1:  PR[91,1] = PR[90,1] + -61.583;
   1:  PR[91,2] = PR[90,2] + 11.317;
   1:L PR[91] R[100]mm/sec CNT100;
   1:  PR[91,1] = PR[90,1] + -63.243;
   1:  PR[91,2] = PR[90,2] + 12.976;
   1:L PR[91] R[100]mm/sec CNT100;
   1:  PR[91,1] = PR[90,1] + -63.972;
   1:  PR[91,2] = PR[90,2] + 13.502;
   1:L PR[91] R[100]mm/sec CNT100;
   1:  PR[91,1] = PR[90,1] + -65.953;
   1:  PR[91,2] = PR[90,2] + 14.889;
   1:L PR[91] R[100]mm/sec CNT100;
   1:  PR[91,1] = PR[90,1] + -68.136;
   1:  PR[91,2] = PR[90,2] + 15.906;
   1:L PR[91] R[100]mm/sec CNT100;
   1:  PR[91,1] = PR[90,1] + -68.941;
   1:  PR[91,2] = PR[90,2] + 16.262;
   1:L PR[91] R[100]mm/sec CNT100;
   1:  PR[91,1] = PR[90,1] + -71.302;
   1:  PR[91,2] = PR[90,2] + 16.894;
   1:L PR[91] R[100]mm/sec CNT100;
   1:  PR[91,1] = PR[90,1] + -72.101;
   1:  PR[91,2] = PR[90,2] + 17.062;
   1:L PR[91] R[100]mm/sec CNT100;
   1:  PR[91,1] = PR[90,1] + -74.577;
   1:  PR[91,2] = PR[90,2] + 17.278;
   1:L PR[91] R[100]mm/sec CNT100;
   1:  PR[91,1] = PR[90,1] + -75.333;
   1:  PR[91,2] = PR[90,2] + 17.277;
   1:L PR[91] R[100]mm/sec CNT100;
   1:  PR[91,1] = PR[90,1] + -77.848;
   1:  PR[91,2] = PR[90,2] + 17.056;
   1:L PR[91] R[100]mm/sec CNT100;
   1:  PR[91,1] = PR[90,1] + -78.535;
   1:  PR[91,2] = PR[90,2] + 16.909;
   1:L PR[91] R[100]mm/sec CNT100;
   1:  PR[91,1] = PR[90,1] + -80.998;
   1:  PR[91,2] = PR[90,2] + 16.248;
   1:L PR[91] R[100]mm/sec CNT100;
   1:  PR[91,1] = PR[90,1] + -83.975;
   1:  PR[91,2] = PR[90,2] + 14.873;
   1:L PR[91] R[100]mm/sec CNT100;
   1:  PR[91,1] = PR[90,1] + -86.111;
   1:  PR[91,2] = PR[90,2] + 13.377;
   1:L PR[91] R[100]mm/sec CNT100;
   1:  PR[91,1] = PR[90,1] + -86.633;
   1:  PR[91,2] = PR[90,2] + 12.996;
   1:L PR[91] R[100]mm/sec CNT100;
   1:  PR[91,1] = PR[90,1] + -88.480;
   1:  PR[91,2] = PR[90,2] + 11.149;
   1:L PR[91] R[100]mm/sec CNT100;
   1:  PR[91,1] = PR[90,1] + -88.889;
   1:  PR[91,2] = PR[90,2] + 10.693;
   1:L PR[91] R[100]mm/sec CNT100;
   1:  PR[91,1] = PR[90,1] + -90.405;
   1:  PR[91,2] = PR[90,2] + 8.528;
   1:L PR[91] R[100]mm/sec CNT100;
   1:  PR[91,1] = PR[90,1] + -90.699;
   1:  PR[91,2] = PR[90,2] + 8.018;
   1:L PR[91] R[100]mm/sec CNT100;
   1:  PR[91,1] = PR[90,1] + -91.818;
   1:  PR[91,2] = PR[90,2] + 5.618;
   1:L PR[91] R[100]mm/sec CNT100;
   1:  PR[91,1] = PR[90,1] + -91.995;
   1:  PR[91,2] = PR[90,2] + 5.073;
   1:L PR[91] R[100]mm/sec CNT100;
   1:  PR[91,1] = PR[90,1] + -92.680;
   1:  PR[91,2] = PR[90,2] + 2.517;
   1:L PR[91] R[100]mm/sec CNT100;
   1:  PR[91,1] = PR[90,1] + -92.915;
   1:  PR[91,2] = PR[90,2] + -0.180;
   1:L PR[91] R[100]mm/sec CNT100;
   1:  PR[91,1] = PR[90,1] + -92.975;
   1:  PR[91,2] = PR[90,2] + -0.747;
   1:L PR[91] R[100]mm/sec CNT100;
   1:  PR[91,1] = PR[90,1] + -92.744;
   1:  PR[91,2] = PR[90,2] + -3.386;
   1:L PR[91] R[100]mm/sec CNT100;
   1:  PR[91,1] = PR[90,1] + -92.680;
   1:  PR[91,2] = PR[90,2] + -3.936;
   1:L PR[91] R[100]mm/sec CNT100;
   1:  PR[91,1] = PR[90,1] + -91.971;
   1:  PR[91,2] = PR[90,2] + -6.581;
   1:L PR[91] R[100]mm/sec CNT100;
   1:  PR[91,1] = PR[90,1] + -91.817;
   1:  PR[91,2] = PR[90,2] + -7.056;
   1:L PR[91] R[100]mm/sec CNT100TB   .50sec,CALL END_PUD;
   1:  PR[92] = PR[91];
   1:  PR[92,3] = PR[92,3] + 20;
   1:J PR[92] 10% FINE;
   1:  PR[91] = PR[90];
   1:  PR[91,1] = PR[90,1] + 19.063;
   1:  PR[91,2] = PR[90,2] + 16.431;
   1:  PR[91,3] = PR[90,3] + 11.895;
   1:  PR[92] = PR[91];
   1:  PR[92,3] = PR[92,3] + 20;
   1:J PR[92] 10% FINE;
   1:L PR[91] R[100]mm/sec CNT100;
   1:  CALL LASER_DRAHT_START;
   1:  PR[91,1] = PR[90,1] + 16.739;
   1:  PR[91,2] = PR[90,2] + 15.346;
   1:L PR[91] R[100]mm/sec CNT100;
   1:  PR[91,1] = PR[90,1] + 15.777;
   1:  PR[91,2] = PR[90,2] + 14.950;
   1:L PR[91] R[100]mm/sec CNT100;
   1:  PR[91,1] = PR[90,1] + 13.786;
   1:  PR[91,2] = PR[90,2] + 13.556;
   1:L PR[91] R[100]mm/sec CNT100;
   1:  PR[91,1] = PR[90,1] + 12.946;
   1:  PR[91,2] = PR[90,2] + 12.913;
   1:L PR[91] R[100]mm/sec CNT100;
   1:  PR[91,1] = PR[90,1] + 11.237;
   1:  PR[91,2] = PR[90,2] + 11.205;
   1:L PR[91] R[100]mm/sec CNT100;
   1:  PR[91,1] = PR[90,1] + 10.585;
   1:  PR[91,2] = PR[90,2] + 10.356;
   1:L PR[91] R[100]mm/sec CNT100;
   1:  PR[91,1] = PR[90,1] + 9.172;
   1:  PR[91,2] = PR[90,2] + 8.338;
   1:L PR[91] R[100]mm/sec CNT100;
   1:  PR[91,1] = PR[90,1] + 8.133;
   1:  PR[91,2] = PR[90,2] + 6.110;
   1:L PR[91] R[100]mm/sec CNT100;
   1:  PR[91,1] = PR[90,1] + 7.721;
   1:  PR[91,2] = PR[90,2] + 5.117;
   1:L PR[91] R[100]mm/sec CNT100;
   1:  PR[91,1] = PR[90,1] + 7.108;
   1:  PR[91,2] = PR[90,2] + 2.826;
   1:L PR[91] R[100]mm/sec CNT100;
   1:  PR[91,1] = PR[90,1] + 6.887;
   1:  PR[91,2] = PR[90,2] + 0.298;
   1:L PR[91] R[100]mm/sec CNT100;
   1:  PR[91,1] = PR[90,1] + 6.747;
   1:  PR[91,2] = PR[90,2] + -0.772;
   1:L PR[91] R[100]mm/sec CNT100;
   1:  PR[91,1] = PR[90,1] + 6.961;
   1:  PR[91,2] = PR[90,2] + -3.220;
   1:L PR[91] R[100]mm/sec CNT100;
   1:  PR[91,1] = PR[90,1] + 7.096;
   1:  PR[91,2] = PR[90,2] + -4.243;
   1:L PR[91] R[100]mm/sec CNT100;
   1:  PR[91,1] = PR[90,1] + 7.721;
   1:  PR[91,2] = PR[90,2] + -6.577;
   1:L PR[91] R[100]mm/sec CNT100;
   1:  PR[91,1] = PR[90,1] + 8.134;
   1:  PR[91,2] = PR[90,2] + -7.570;
   1:L PR[91] R[100]mm/sec CNT100;
   1:  PR[91,1] = PR[90,1] + 9.173;
   1:  PR[91,2] = PR[90,2] + -9.799;
   1:L PR[91] R[100]mm/sec CNT100;
   1:  PR[91,1] = PR[90,1] + 10.587;
   1:  PR[91,2] = PR[90,2] + -11.817;
   1:L PR[91] R[100]mm/sec CNT100;
   1:  PR[91,1] = PR[90,1] + 11.240;
   1:  PR[91,2] = PR[90,2] + -12.667;
   1:L PR[91] R[100]mm/sec CNT100;
   1:  PR[91,1] = PR[90,1] + 12.950;
   1:  PR[91,2] = PR[90,2] + -14.375;
   1:L PR[91] R[100]mm/sec CNT100;
   1:  PR[91,1] = PR[90,1] + 13.790;
   1:  PR[91,2] = PR[90,2] + -15.018;
   1:L PR[91] R[100]mm/sec CNT100;
   1:  PR[91,1] = PR[90,1] + 15.820;
   1:  PR[91,2] = PR[90,2] + -16.438;
   1:L PR[91] R[100]mm/sec CNT100;
   1:  PR[91,1] = PR[90,1] + 18.057;
   1:  PR[91,2] = PR[90,2] + -17.480;
   1:L PR[91] R[100]mm/sec CNT100;
   1:  PR[91,1] = PR[90,1] + 19.027;
   1:  PR[91,2] = PR[90,2] + -17.880;
   1:L PR[91] R[100]mm/sec CNT100;
   1:  PR[91,1] = PR[90,1] + 21.383;
   1:  PR[91,2] = PR[90,2] + -18.511;
   1:L PR[91] R[100]mm/sec CNT100;
   1:  PR[91,1] = PR[90,1] + 22.407;
   1:  PR[91,2] = PR[90,2] + -18.644;
   1:L PR[91] R[100]mm/sec CNT100;
   1:  PR[91,1] = PR[90,1] + 24.887;
   1:  PR[91,2] = PR[90,2] + -18.860;
   1:L PR[91] R[100]mm/sec CNT100;
   1:  PR[91,1] = PR[90,1] + 27.363;
   1:  PR[91,2] = PR[90,2] + -18.643;
   1:L PR[91] R[100]mm/sec CNT100;
   1:  PR[91,1] = PR[90,1] + 28.377;
   1:  PR[91,2] = PR[90,2] + -18.507;
   1:L PR[91] R[100]mm/sec CNT100;
   1:  PR[91,1] = PR[90,1] + 30.707;
   1:  PR[91,2] = PR[90,2] + -17.882;
   1:L PR[91] R[100]mm/sec CNT100;
   1:  PR[91,1] = PR[90,1] + 33.043;
   1:  PR[91,2] = PR[90,2] + -16.793;
   1:L PR[91] R[100]mm/sec CNT100;
   1:  PR[91,1] = PR[90,1] + 33.979;
   1:  PR[91,2] = PR[90,2] + -16.403;
   1:L PR[91] R[100]mm/sec CNT100;
   1:  PR[91,1] = PR[90,1] + 35.997;
   1:  PR[91,2] = PR[90,2] + -14.989;
   1:L PR[91] R[100]mm/sec CNT100;
   1:  PR[91,1] = PR[90,1] + 36.789;
   1:  PR[91,2] = PR[90,2] + -14.380;
   1:L PR[91] R[100]mm/sec CNT100;
   1:  PR[91,1] = PR[90,1] + 38.531;
   1:  PR[91,2] = PR[90,2] + -12.639;
   1:L PR[91] R[100]mm/sec CNT100;
   1:  PR[91,1] = PR[90,1] + 39.131;
   1:  PR[91,2] = PR[90,2] + -11.855;
   1:L PR[91] R[100]mm/sec CNT100;
   1:  PR[91,1] = PR[90,1] + 40.578;
   1:  PR[91,2] = PR[90,2] + -9.789;
